# B&R Automation Studio project MotionTestBenchMaster (part 38)

#### Cyclic.sfc - Cyclic code
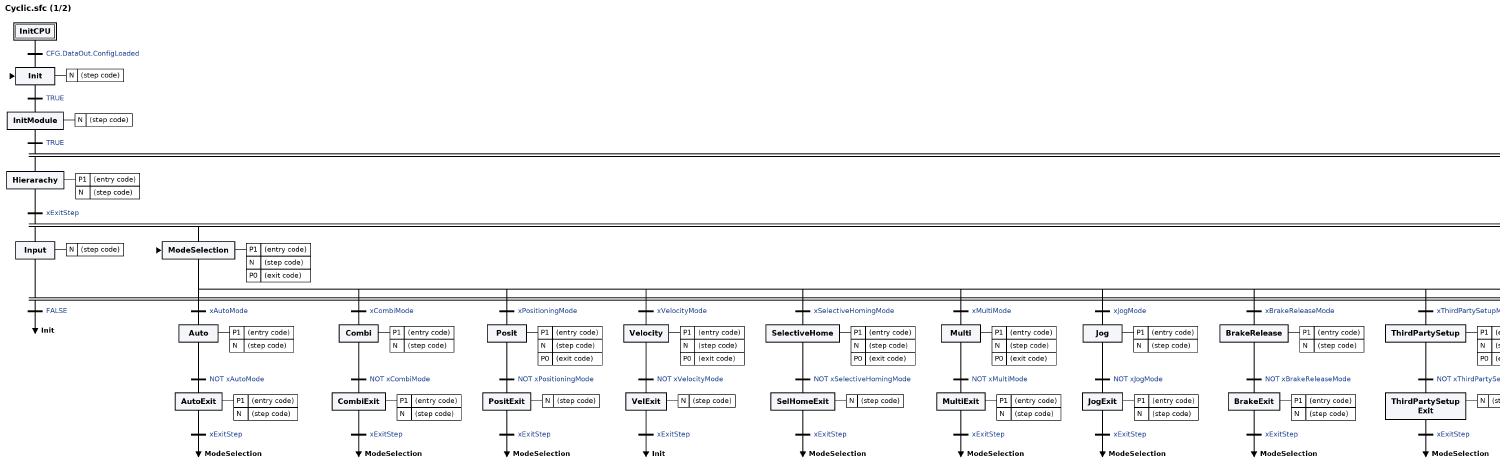
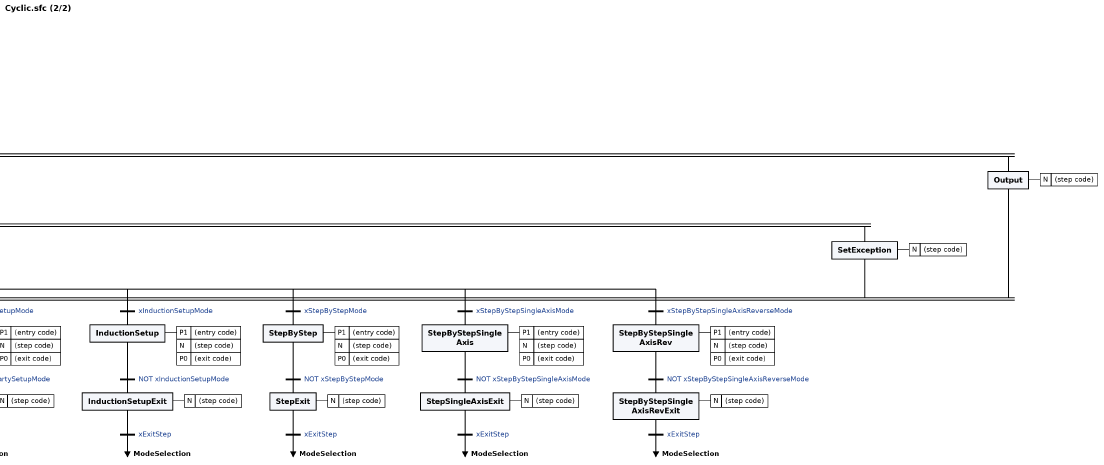
```iecst
PROGRAM _CYCLIC
INITIAL_STEP InitCPU:
END_STEP
TRANSITION FROM InitCPU TO Init:=
CFG.DataOut.ConfigLoaded
END_TRANSITION
STEP Init:
(* Pointer to master position *)
IF NOT CFG_MC.Generic.SyncroPar.ExternalEncoder THEN
	VAR_Machine.stMasterModule.iq_stParameters.i_pstMasterPositionStruct	:= ADR(ITC_Motion);	//VIRTUAL POSITION (SUPERCOMBI)
END_IF

// Init Encoder Emulation
fbEncoderEmulation.i_pstSrcAxis			:= ADR(VAR_AxFillerMain);
fbEncoderEmulation.i_pstEncEmulAxis		:= ADR(VAR_AxEncEmul);
IF CFG_MC.Generic.EmulationCardPulses > 0 THEN
	fbEncoderEmulation.i_uiNumberOfPulses	:= CFG_MC.Generic.EmulationCardPulses;
ELSE
	fbEncoderEmulation.i_uiNumberOfPulses	:= 1024;
END_IF
fbEncoderEmulation.i_xEnable			:= TRUE;
END_STEP
TRANSITION FROM Init TO InitModule:=
TRUE
END_TRANSITION
STEP InitModule:
MC_InputOutput;

(* Machine excpetion *)
fbQuickStopFromPlc.i_psAlarmName		:= ADR('PlcQuickStop');
fbQuickStopFromPlc.i_pstMpAlarmXLink	:= ADR(gMainAlarmXCoreLink);
fbQuickStopFromPlc.i_pxAcknowledge		:= ADR(VAR_Machine.iq_stCmd.i_xReset);
fbQuickStopFromPlc.i_pxInitCoreDone		:= ADR(VAR_Machine.stMasterModule.iq_stCmd.i_xAlarmInitOk);
fbQuickStopFromPlc.i_xAutoAck			:= TRUE;

fbKochModuleNotReady.i_psAlarmName		:= ADR('KochNotReady');
fbKochModuleNotReady.i_pstMpAlarmXLink	:= ADR(gMainAlarmXCoreLink);
fbKochModuleNotReady.i_pxAcknowledge	:= ADR(VAR_Machine.iq_stCmd.i_xReset);
fbKochModuleNotReady.i_pxInitCoreDone	:= ADR(VAR_Machine.stMasterModule.iq_stCmd.i_xAlarmInitOk);
fbKochModuleNotReady.i_xAutoAck			:= TRUE;

fbSeamerFanFault.i_psAlarmName			:= ADR('SeamerFanFault');
fbSeamerFanFault.i_pstMpAlarmXLink		:= ADR(gMainAlarmXCoreLink);
fbSeamerFanFault.i_pxAcknowledge		:= ADR(VAR_Machine.iq_stCmd.i_xReset);
fbSeamerFanFault.i_pxInitCoreDone		:= ADR(VAR_Machine.stMasterModule.iq_stCmd.i_xAlarmInitOk);
fbSeamerFanFault.i_xAutoAck				:= FALSE;
END_STEP
TRANSITION FROM InitModule TO (Hierarachy,Output):=
TRUE
END_TRANSITION
STEP Hierarachy:
IF 	VAR_Machine.stFillerModule.iq_stStatus.q_xInitDone	AND
	VAR_Machine.stInletModule.iq_stStatus.q_xInitDone 	AND
	VAR_Machine.stOutletModule.iq_stStatus.q_xInitDone	THEN

	xExitStep	:=	TRUE;

	// First and last real FILLER axis
	uiMinRealFillerIndex := CST_LastFillerModuleAxis;
	uiMaxRealFillerIndex := CST_FirstFillerModuleAxis;

	FOR uiAxisIndex := CST_FirstFillerModuleAxis TO CST_LastFillerModuleAxis DO
		IF VAR_Machine.stFillerModule.iq_astSubModuleAxis[uiAxisIndex].iq_stStatus.q_stMainAxisStatus.q_xAxisReal THEN
			uiMinRealFillerIndex := MIN(uiMinRealFillerIndex, uiAxisIndex);
			uiMaxRealFillerIndex := MAX(uiMaxRealFillerIndex, uiAxisIndex);
		END_IF
	END_FOR

	// Inlet module last axis homing position = filler module first axis act position
	uiMaxRealInletIndex := CST_FirstInletModuleAxis;
	IF VAR_Machine.stInletModule.iq_stStatus.q_xModuleReal	THEN
		FOR uiAxisIndex := CST_MainAxis TO CST_LastInletModuleAxis DO
			IF VAR_Machine.stInletModule.iq_astSubModuleAxis[uiAxisIndex].iq_stStatus.q_stMainAxisStatus.q_xAxisReal THEN
				uiMaxRealInletIndex := MAX(uiMaxRealInletIndex, uiAxisIndex);
			END_IF
		END_FOR
		IF uiMaxRealInletIndex <> CST_FirstInletModuleAxis THEN
			VAR_Machine.stInletModule.iq_astSubModuleAxis[uiMaxRealInletIndex].iq_stParam.i_udiHomingPosition	:=
				ADR(VAR_Machine.stFillerModule.iq_astSubModuleAxis[uiMinRealFillerIndex].iq_stStatus.q_stMainAxisStatus.q_lrPosition);
		END_IF
	END_IF

	// Outlet module first axis homing position = filler module last axis act position
	uiMinRealOutletIndex := CST_LastOutletModuleAxis;
	IF VAR_Machine.stOutletModule.iq_stStatus.q_xModuleReal	THEN
		FOR uiAxisIndex := CST_FirstOutletModuleAxis TO CST_MainAxis DO
			IF VAR_Machine.stOutletModule.iq_astSubModuleAxis[uiAxisIndex].iq_stStatus.q_stMainAxisStatus.q_xAxisReal THEN
				uiMinRealOutletIndex := MIN(uiMinRealOutletIndex, uiAxisIndex);
			END_IF
		END_FOR
		IF uiMinRealOutletIndex <> CST_LastOutletModuleAxis THEN
			VAR_Machine.stOutletModule.iq_astSubModuleAxis[uiMinRealOutletIndex].iq_stParam.i_udiHomingPosition	:=
				ADR(VAR_Machine.stFillerModule.iq_astSubModuleAxis[uiMaxRealFillerIndex].iq_stStatus.q_stMainAxisStatus.q_lrPosition);
		END_IF
	END_IF
END_IF

//NEW MANAGEMENT //FR
HMI_AxisIndex := 2;//0 is master
//HMI Crate array axis present and name
//INlet Module
IF VAR_Machine.stInletModule.iq_stStatus.q_xModuleReal THEN
	FOR uiAxisIndex := CST_FirstInletModuleAxis TO CST_LastInletModuleAxis DO
		IF VAR_Machine.stInletModule.iq_astSubModuleAxis[uiAxisIndex].iq_stStatus.q_stMainAxisStatus.q_xAxisReal THEN
			HMI_MC_GenericAxisDataNew[HMI_AxisIndex].xHmiPresent	:= TRUE;
			HMI_MC_GenericAxisDataNew[HMI_AxisIndex].uiAxisID		:= uiAxisIndex + CST_InletSubModuleHmiStart;
			HMI_AxisIndex := HMI_AxisIndex +1;
		END_IF
	END_FOR
END_IF
//HMI Crate array axis present and name
//Filler Module
IF VAR_Machine.stFillerModule.iq_stStatus.q_xModuleReal	THEN
	FOR uiAxisIndex := CST_FirstFillerModuleAxis TO CST_LastFillerModuleAxis DO
		IF VAR_Machine.stFillerModule.iq_astSubModuleAxis[uiAxisIndex].iq_stStatus.q_stMainAxisStatus.q_xAxisReal THEN
			HMI_MC_GenericAxisDataNew[HMI_AxisIndex].xHmiPresent	:= TRUE;
			HMI_MC_GenericAxisDataNew[HMI_AxisIndex].uiAxisID		:= uiAxisIndex + CST_FillerSubModuleHmiStart;
			HMI_AxisIndex := HMI_AxisIndex +1;
		END_IF
	END_FOR
END_IF
//HMI Crate array axis present and name
//Outlet Module
IF VAR_Machine.stOutletModule.iq_stStatus.q_xModuleReal	THEN
	FOR uiAxisIndex := CST_FirstOutletModuleAxis TO CST_LastOutletModuleAxis DO
		IF VAR_Machine.stOutletModule.iq_astSubModuleAxis[uiAxisIndex].iq_stStatus.q_stMainAxisStatus.q_xAxisReal THEN
			HMI_MC_GenericAxisDataNew[HMI_AxisIndex].xHmiPresent	:= TRUE;
			HMI_MC_GenericAxisDataNew[HMI_AxisIndex].uiAxisID		:= uiAxisIndex + CST_OutletSubModuleHmiStart;
			HMI_AxisIndex := HMI_AxisIndex +1;
		END_IF
	END_FOR
END_IF

FOR HMI_AxisIndex := 2 TO 14 DO //vrma

CASE HMI_MC_GenericAxisDataNew[HMI_AxisIndex].uiAxisID OF

	105:
		HMI_MC_GenericAxisDataNew[HMI_AxisIndex].usiHmiName	:= CFG_MC.Axes.Filler.In[10].HmiNameId;

	106:
		HMI_MC_GenericAxisDataNew[HMI_AxisIndex].usiHmiName	:= CFG_MC.Axes.Filler.In[9].HmiNameId;

	107:
		HMI_MC_GenericAxisDataNew[HMI_AxisIndex].usiHmiName	:= CFG_MC.Axes.Filler.In[8].HmiNameId;

	108:
		HMI_MC_GenericAxisDataNew[HMI_AxisIndex].usiHmiName	:= CFG_MC.Axes.Filler.In[7].HmiNameId;

	109:
		HMI_MC_GenericAxisDataNew[HMI_AxisIndex].usiHmiName	:= CFG_MC.Axes.Filler.In[6].HmiNameId;

	110:
		HMI_MC_GenericAxisDataNew[HMI_AxisIndex].usiHmiName	:= CFG_MC.Axes.Filler.In[5].HmiNameId;

	111:
		HMI_MC_GenericAxisDataNew[HMI_AxisIndex].usiHmiName	:= CFG_MC.Axes.Filler.In[4].HmiNameId;

	112:
		HMI_MC_GenericAxisDataNew[HMI_AxisIndex].usiHmiName	:= CFG_MC.Axes.Filler.In[3].HmiNameId;

	113:
		HMI_MC_GenericAxisDataNew[HMI_AxisIndex].usiHmiName	:= CFG_MC.Axes.Filler.In[2].HmiNameId;

	114:
		HMI_MC_GenericAxisDataNew[HMI_AxisIndex].usiHmiName	:= CFG_MC.Axes.Filler.In[1].HmiNameId;

	115:
		HMI_MC_GenericAxisDataNew[HMI_AxisIndex].usiHmiName	:= CFG_MC.Axes.Filler.Main.HmiNameId;

	116:
		HMI_MC_GenericAxisDataNew[HMI_AxisIndex].usiHmiName	:= CFG_MC.Axes.Filler.Out[1].HmiNameId;

	117:
		HMI_MC_GenericAxisDataNew[HMI_AxisIndex].usiHmiName	:= CFG_MC.Axes.Filler.Out[2].HmiNameId;

	118:
		HMI_MC_GenericAxisDataNew[HMI_AxisIndex].usiHmiName	:= CFG_MC.Axes.Filler.Out[3].HmiNameId;

	119:
		HMI_MC_GenericAxisDataNew[HMI_AxisIndex].usiHmiName	:= CFG_MC.Axes.Filler.Out[4].HmiNameId;

	120:
		HMI_MC_GenericAxisDataNew[HMI_AxisIndex].usiHmiName	:= CFG_MC.Axes.Filler.Out[5].HmiNameId;

	121:
		HMI_MC_GenericAxisDataNew[HMI_AxisIndex].usiHmiName	:= CFG_MC.Axes.Filler.Out[6].HmiNameId;

	211:
		HMI_MC_GenericAxisDataNew[HMI_AxisIndex].usiHmiName	:= CFG_MC.Axes.Inlet.In[4].HmiNameId;

	212:
		HMI_MC_GenericAxisDataNew[HMI_AxisIndex].usiHmiName	:= CFG_MC.Axes.Inlet.In[3].HmiNameId;

	213:
		HMI_MC_GenericAxisDataNew[HMI_AxisIndex].usiHmiName	:= CFG_MC.Axes.Inlet.In[2].HmiNameId;

	214:
		HMI_MC_GenericAxisDataNew[HMI_AxisIndex].usiHmiName	:= CFG_MC.Axes.Inlet.In[1].HmiNameId;

	215:
		HMI_MC_GenericAxisDataNew[HMI_AxisIndex].usiHmiName	:= CFG_MC.Axes.Inlet.Main.HmiNameId;

	216:
		HMI_MC_GenericAxisDataNew[HMI_AxisIndex].usiHmiName	:= CFG_MC.Axes.Inlet.Out[1].HmiNameId;

	217:
		HMI_MC_GenericAxisDataNew[HMI_AxisIndex].usiHmiName	:= CFG_MC.Axes.Inlet.Out[2].HmiNameId;

	218:
		HMI_MC_GenericAxisDataNew[HMI_AxisIndex].usiHmiName	:= CFG_MC.Axes.Inlet.Out[3].HmiNameId;

	219:
		HMI_MC_GenericAxisDataNew[HMI_AxisIndex].usiHmiName	:= CFG_MC.Axes.Inlet.Out[4].HmiNameId;

	311:
		HMI_MC_GenericAxisDataNew[HMI_AxisIndex].usiHmiName	:= CFG_MC.Axes.Outlet.In[4].HmiNameId;

	312:
		HMI_MC_GenericAxisDataNew[HMI_AxisIndex].usiHmiName	:= CFG_MC.Axes.Outlet.In[3].HmiNameId;

	313:
		HMI_MC_GenericAxisDataNew[HMI_AxisIndex].usiHmiName	:= CFG_MC.Axes.Outlet.In[2].HmiNameId;

	314:
		HMI_MC_GenericAxisDataNew[HMI_AxisIndex].usiHmiName	:= CFG_MC.Axes.Outlet.In[1].HmiNameId;

	315:
		HMI_MC_GenericAxisDataNew[HMI_AxisIndex].usiHmiName	:= CFG_MC.Axes.Outlet.Main.HmiNameId;

	316:
		HMI_MC_GenericAxisDataNew[HMI_AxisIndex].usiHmiName	:= CFG_MC.Axes.Outlet.Out[1].HmiNameId;

	317:
		HMI_MC_GenericAxisDataNew[HMI_AxisIndex].usiHmiName	:= CFG_MC.Axes.Outlet.Out[2].HmiNameId;

	318:
		HMI_MC_GenericAxisDataNew[HMI_AxisIndex].usiHmiName	:= CFG_MC.Axes.Outlet.Out[3].HmiNameId;

	319:
		HMI_MC_GenericAxisDataNew[HMI_AxisIndex].usiHmiName	:= CFG_MC.Axes.Outlet.Out[4].HmiNameId;
	ELSE
		HMI_MC_GenericAxisDataNew[HMI_AxisIndex].usiHmiName		:= 0;
END_CASE

END_FOR
END_STEP
ENTRY_ACTION
xExitStep	:=	FALSE;

VAR_Machine.stMasterModule.iq_stCmd.i_xMachineInitDone	:=	TRUE;
VAR_Machine.stFillerModule.iq_stCmd.i_xMachineInitDone	:=	TRUE;
VAR_Machine.stInletModule.iq_stCmd.i_xMachineInitDone	:=	TRUE;
VAR_Machine.stOutletModule.iq_stCmd.i_xMachineInitDone	:=	TRUE;
END_ACTION
TRANSITION FROM Hierarachy TO (Input,ModeSelection,SetException):=
xExitStep
END_TRANSITION
STEP Input:
(* Input Signals *)
xInputJog							:= VAR_Machine.iq_stCmd.i_xJogMode;
xInputAuto							:= VAR_Machine.iq_stCmd.i_xAuto	AND NOT VAR_Machine.iq_stCmd.i_xStepByStep AND NOT VAR_Machine.iq_stCmd.i_xStepByStepSingleAxis AND NOT VAR_Machine.iq_stCmd.i_xStepByStepSingleAxisReverse;//v999
xInputCombi							:= VAR_Machine.iq_stCmd.i_xCombi;
xInputMulti							:= VAR_Machine.iq_stCmd.i_xMulti;
xInputSelHoming						:= VAR_Machine.iq_stCmd.i_xSelectiveHoming;
xInputPositioning					:= VAR_Machine.iq_stCmd.i_xPositioning;
xInputBrakeRelease					:= VAR_Machine.iq_stCmd.i_xBrakeRelease;
xInputVelocity						:= VAR_Machine.iq_stCmd.i_xVelocity;
xInputStepByStep					:= VAR_Machine.iq_stCmd.i_xAuto AND VAR_Machine.iq_stCmd.i_xStepByStep;
xInputStepByStepSingleAxis			:= (VAR_Machine.iq_stCmd.i_xAuto AND VAR_Machine.iq_stCmd.i_xStepByStepSingleAxis) OR (NOT VAR_Machine.iq_stCmd.i_xAuto AND VAR_Machine.iq_stCmd.i_xStepByStepSingleAxis);//V4.A.A.1.7.0 FootBar
xInputStepByStepSingleAxisRev		:= (VAR_Machine.iq_stCmd.i_xAuto AND VAR_Machine.iq_stCmd.i_xStepByStepSingleAxisReverse) OR (NOT VAR_Machine.iq_stCmd.i_xAuto AND VAR_Machine.iq_stCmd.i_xStepByStepSingleAxisReverse);//v999
xInputThirdPartySetup				:= VAR_Machine.iq_stCmd.i_xThirdPartySetup;
xInputInductionSetup				:= VAR_Machine.iq_stCmd.i_xInductionSetup;

(* Acceleration and deceleration calculation *)
IF 	rOldAccelerationValue <> MC_InputOutput.Network.Machine.Parameters.AutoAccelerationTime 	AND
	MC_InputOutput.Network.Machine.Parameters.AutoAccelerationTime > 0						  	AND
	MC_InputOutput.Network.Machine.Status.MachineMaxSpeed	> 0									THEN

	VAR_Machine.stMasterModule.iq_stParameters.i_rEndlessAcceleration
		:= FC_GetAccFromTimeAndJerk(	MC_InputOutput.Network.Machine.Parameters.AutoAccelerationTime,
								 		CFG_MC.Movements.Jerk,
										MC_InputOutput.Network.Machine.Status.MachineMaxSpeed / 10.0);

	VAR_Machine.stMasterModule.iq_stParameters.i_rEndlessAcceleration
		:= MIN(VAR_Machine.stMasterModule.iq_stParameters.i_rEndlessAcceleration, VAR_EmergencyDec);

	VAR_Machine.stFillerModule.iq_stParameters.i_rEndlessAcceleration
		:= VAR_Machine.stMasterModule.iq_stParameters.i_rEndlessAcceleration;

	VAR_Machine.stInletModule.iq_stParameters.i_rEndlessAcceleration
		:= VAR_Machine.stMasterModule.iq_stParameters.i_rEndlessAcceleration;

	VAR_Machine.stOutletModule.iq_stParameters.i_rEndlessAcceleration
		:= VAR_Machine.stMasterModule.iq_stParameters.i_rEndlessAcceleration;

	rOldAccelerationValue := MC_InputOutput.Network.Machine.Parameters.AutoAccelerationTime;
END_IF

IF 	rOldDecelerationValue <> MC_InputOutput.Network.Machine.Parameters.AutoDecelerationTime 	AND
	MC_InputOutput.Network.Machine.Parameters.AutoDecelerationTime 	> 0					  		AND
	MC_InputOutput.Network.Machine.Status.MachineMaxSpeed			> 0							THEN

	VAR_Machine.stMasterModule.iq_stParameters.i_rEndlessDeceleration
		:= FC_GetAccFromTimeAndJerk(	MC_InputOutput.Network.Machine.Parameters.AutoDecelerationTime,
										CFG_MC.Movements.Jerk,
										MC_InputOutput.Network.Machine.Status.MachineMaxSpeed / 10.0);

	VAR_Machine.stMasterModule.iq_stParameters.i_rEndlessDeceleration
		:= MIN(VAR_Machine.stMasterModule.iq_stParameters.i_rEndlessDeceleration, VAR_EmergencyDec);

	VAR_Machine.stFillerModule.iq_stParameters.i_rEndlessDeceleration
		:= VAR_Machine.stMasterModule.iq_stParameters.i_rEndlessDeceleration;

	VAR_Machine.stInletModule.iq_stParameters.i_rEndlessDeceleration
		:= VAR_Machine.stMasterModule.iq_stParameters.i_rEndlessDeceleration;

	VAR_Machine.stOutletModule.iq_stParameters.i_rEndlessDeceleration
		:= VAR_Machine.stMasterModule.iq_stParameters.i_rEndlessDeceleration;

	rOldDecelerationValue := MC_InputOutput.Network.Machine.Parameters.AutoDecelerationTime;
END_IF

(* Enable curves *)
VAR_Machine.stMasterModule.iq_stCmd.i_xEnableCurves	:=	MC_InputOutput.Network.Machine.Commands.MasterEncoderPositionValid; //COMBI

(* Input from safety system *)
VAR_Machine.stFillerModule.iq_stCmd.i_xEnable	:= MC_InputOutput.Safety.Filler.Commands.EnableModule;
VAR_Machine.stInletModule.iq_stCmd.i_xEnable	:= MC_InputOutput.Safety.Inlet.Commands.EnableModule;
VAR_Machine.stOutletModule.iq_stCmd.i_xEnable	:= MC_InputOutput.Safety.Outlet.Commands.EnableModule;

xSlowMotionCommandOutletForward		:= MC_InputOutput.Network.Outlet.Commands.SlowMotionForward;
xSlowMotionCommandOutletBackward	:= MC_InputOutput.Network.Outlet.Commands.SlowMotionBackward;
xSlowMotionCommandOutlet			:= xSlowMotionCommandOutletForward OR xSlowMotionCommandOutletBackward;

xSlowMotionCommandInletForward		:= MC_InputOutput.Network.Inlet.Commands.SlowMotionForward;
xSlowMotionCommandInletBackward		:= MC_InputOutput.Network.Inlet.Commands.SlowMotionBackward;
xSlowMotionCommandInlet				:= xSlowMotionCommandInletForward OR xSlowMotionCommandInletBackward;
END_STEP
STEP ModeSelection:
xModeReady	:= NOT xAutoMode AND NOT xPositioningMode AND NOT xSelectiveHomingMode	AND NOT xJogMode AND NOT xPositioningMode AND NOT xThirdPartySetupMode AND NOT xInductionSetupMode AND
				(NOT tofReactionActive.Q OR	xInputMulti OR xInputStepByStepSingleAxis);//V1.7.2

xNoOpActive				:= TRUE;
xAutoActive				:= FALSE;
xBrakeReleaseActive		:= FALSE;
xPositioningActive		:= FALSE;
xSelHomingActive		:= FALSE;
xJogActive				:= FALSE;
xMultiActive			:= FALSE;
xVelocityActive			:= FALSE;
xStepByStepActive		:= FALSE;
xStepByStepSingleAxisActive	:= FALSE;//V4.A.A.1.7.0
xStepByStepSingleAxisRevActive	:= FALSE; //v999
xCombiActive			:= FALSE;
xThirdPartySetupActive	:= FALSE;
xInductionSetupActive	:= FALSE;

IF xModeReady THEN
	IF xInputAuto THEN
		xAutoMode					:= TRUE;
	ELSIF xInputCombi THEN
		xCombiMode					:= TRUE;
	ELSIF xInputPositioning THEN
		xPositioningMode			:= TRUE;
	ELSIF xInputSelHoming THEN
		xSelectiveHomingMode		:= TRUE;
	ELSIF xInputJog THEN
		xJogMode					:= TRUE;
	ELSIF xInputMulti THEN
		xMultiMode					:= TRUE;
	ELSIF xInputVelocity THEN
		xVelocityMode				:= TRUE;
	ELSIF xInputStepByStep THEN
		xStepByStepMode				:= TRUE;
	ELSIF xInputStepByStepSingleAxis THEN//V4.A.A.1.7.0
		xStepByStepSingleAxisMode	:= TRUE;//V4.A.A.1.7.0
	ELSIF xInputStepByStepSingleAxisRev THEN//v999
		xStepByStepSingleAxisReverseMode := TRUE;//v999
	ELSIF xInputThirdPartySetup THEN
		xThirdPartySetupMode		:= TRUE;
	ELSIF xInputInductionSetup THEN
		xInductionSetupMode			:= TRUE;
	END_IF
ELSIF tofReactionActive.Q AND xInputBrakeRelease THEN
	xBrakeReleaseMode			:= TRUE;
END_IF
END_STEP
ENTRY_ACTION
xExitStep	:= FALSE;

VAR_Machine.stMasterModule.iq_stCmd.i_xStart	:= FALSE;
VAR_Machine.stFillerModule.iq_stCmd.i_xStart	:= FALSE;
VAR_Machine.stInletModule.iq_stCmd.i_xStart		:= FALSE;
VAR_Machine.stOutletModule.iq_stCmd.i_xStart	:= FALSE;

// For safety reason all bits are set to FALSE
xJogMode 							:= FALSE;
xAutoMode 							:= FALSE;
xMultiMode 							:= FALSE;
xPositioningMode 					:= FALSE;
xSelectiveHomingMode				:= FALSE;
xVelocityMode						:= FALSE;
xCombiMode							:= FALSE;
xBrakeReleaseMode					:= FALSE;
xStepByStepMode						:= FALSE;
xStepByStepSingleAxisMode			:= FALSE;//V4.A.A.1.7.0 Footbar
xStepByStepSingleAxisReverseMode	:= FALSE;//V999
xThirdPartySetupMode				:= FALSE;
xInductionSetupMode					:= FALSE;
END_ACTION
EXIT_ACTION
xNoOpActive	:= FALSE;
END_ACTION
TRANSITION FROM ModeSelection TO Auto:=
xAutoMode
END_TRANSITION
TRANSITION FROM ModeSelection TO Combi:=
xCombiMode
END_TRANSITION
STEP Combi:
IF xReactionActive	OR NOT xInputCombi	THEN
	xCombiMode	:=	FALSE;
END_IF

xCombiActive	:= TRUE;

CASE uiCombiStep OF
	0:
		xCombiSynchronized		:=	FALSE;
		xCombiSynchroStopDone	:=	FALSE;
		xCombiFixedSpeed		:=	FALSE;
		xCombiSynchroInProgress	:=	FALSE;

		VAR_Machine.stFillerModule.iq_stCmd.i_xAutoMode	:=	TRUE;
		VAR_Machine.stOutletModule.iq_stCmd.i_xAutoMode	:=	VAR_Machine.stOutletModule.iq_stStatus.q_xModuleReal;
		VAR_Machine.stInletModule.iq_stCmd.i_xAutoMode	:=	VAR_Machine.stInletModule.iq_stStatus.q_xModuleReal;

		uiCombiStep	:=	40;

	40:
		IF 	VAR_Machine.stFillerModule.iq_stStatus.q_xAutoActive	AND
			(VAR_Machine.stOutletModule.iq_stStatus.q_xAutoActive	OR NOT
			VAR_Machine.stOutletModule.iq_stStatus.q_xModuleReal)	AND
			(VAR_Machine.stInletModule.iq_stStatus.q_xAutoActive	OR NOT
			VAR_Machine.stInletModule.iq_stStatus.q_xModuleReal)	THEN

			IF 	NOT VAR_Machine.stFillerModule.iq_stStatus.q_xSynchroWithOffset		AND
				NOT VAR_Machine.stOutletModule.iq_stStatus.q_xSynchroWithOffset		AND
				NOT VAR_Machine.stInletModule.iq_stStatus.q_xSynchroWithOffset		THEN

				VAR_Machine.stMasterModule.iq_stParameters.i_lrRephasingPosition	:=
					FC_RephasingMachine(iq_astInletSubModuleAxis	:=	VAR_Machine.stInletModule.iq_astSubModuleAxis,
										iq_astFillerSubModuleAxis	:=	VAR_Machine.stFillerModule.iq_astSubModuleAxis,
										iq_astOutletSubModuleAxis	:=	VAR_Machine.stOutletModule.iq_astSubModuleAxis);

				VAR_Machine.stFillerModule.iq_stParameters.i_lrRephasingPosition
					:=	VAR_Machine.stMasterModule.iq_stParameters.i_lrRephasingPosition;

				VAR_Machine.stOutletModule.iq_stParameters.i_lrRephasingPosition
					:=	VAR_Machine.stMasterModule.iq_stParameters.i_lrRephasingPosition;

				VAR_Machine.stInletModule.iq_stParameters.i_lrRephasingPosition
					:=	VAR_Machine.stMasterModule.iq_stParameters.i_lrRephasingPosition;

				uiCombiStep	:=	100;
			END_IF
		END_IF

	100:(* Wait Master Rephased *)
		VAR_Machine.stMasterModule.iq_stCmd.i_xCombi					:=	TRUE;
		VAR_Machine.stMasterModule.iq_stCmd.i_xMasterRephasingRequest	:= 	TRUE;

		IF VAR_Machine.stMasterModule.iq_stStatus.q_xCombiActive AND VAR_Machine.stMasterModule.iq_stStatus.q_xMasterRephased THEN
			VAR_Machine.stMasterModule.iq_stCmd.i_xMasterRephasingRequest	:= 	FALSE;
			uiCombiStep	:=	110;
		END_IF

	110:(* Wait for start Signal *)
		IF VAR_Machine.iq_stCmd.i_xStart THEN
			VAR_Machine.stFillerModule.iq_stCmd.i_xStart	:=	TRUE;
			VAR_Machine.stOutletModule.iq_stCmd.i_xStart	:=	VAR_Machine.stOutletModule.iq_stStatus.q_xModuleReal;
			VAR_Machine.stInletModule.iq_stCmd.i_xStart		:=	VAR_Machine.stInletModule.iq_stStatus.q_xModuleReal;
			uiCombiStep	:=	120;
		END_IF

	120:(* Wait for submodules synchronized *)
		IF VAR_Machine.stFillerModule.iq_stStatus.q_xRealAxesSynchronized		AND
			VAR_Machine.stFillerModule.iq_stStatus.q_xAutoActive				AND
			VAR_Machine.stFillerModule.iq_stStatus.q_xMasterRephased			AND

			((VAR_Machine.stOutletModule.iq_stStatus.q_xRealAxesSynchronized	AND
			VAR_Machine.stOutletModule.iq_stStatus.q_xMasterRephased			AND
			VAR_Machine.stOutletModule.iq_stStatus.q_xAutoActive)				OR NOT
			VAR_Machine.stOutletModule.iq_stStatus.q_xModuleReal)				AND

			((VAR_Machine.stInletModule.iq_stStatus.q_xRealAxesSynchronized		AND
			VAR_Machine.stInletModule.iq_stStatus.q_xMasterRephased				AND
			VAR_Machine.stInletModule.iq_stStatus.q_xAutoActive)				OR NOT
			VAR_Machine.stInletModule.iq_stStatus.q_xModuleReal)				THEN

			VAR_Machine.stMasterModule.iq_stCmd.i_xStart	:=	TRUE;
			xEncEmulationEnable	:= TRUE;
			uiCombiStep	:=	130;
		END_IF

	130:(* Wait for master synchronized with the external reference *)
		xCombiSynchroInProgress	:=	TRUE;

		IF NOT VAR_Machine.iq_stCmd.i_xStart THEN
			VAR_Machine.stMasterModule.iq_stCmd.i_xCombiSynchroStop	:=	TRUE;
			uiCombiStep	:=	150;
		ELSIF VAR_Machine.stMasterModule.iq_stStatus.q_xModuleSynchronized THEN
			uiCombiStep	:=	140;
		END_IF

	140:(* Module synchronized with the master *)
		xCombiSynchroInProgress	:=	FALSE;
		xCombiSynchronized		:=	TRUE;
		xCombiSynchroStopDone	:=	FALSE;
		xCombiFixedSpeed		:=	FALSE;

		IF NOT VAR_Machine.iq_stCmd.i_xStart OR VAR_Machine.iq_stCmd.i_xCombiSynchroStop THEN
			xCombiSynchroInProgress	:=	FALSE;
			xCombiSynchronized		:=	FALSE;
			xCombiSynchroStopDone	:=	TRUE;
			xCombiFixedSpeed		:=	FALSE;

			VAR_Machine.stMasterModule.iq_stCmd.i_xCombiSynchroStop	:=	TRUE;
			uiCombiStep		:=	150;
		ELSIF VAR_Machine.iq_stCmd.i_xOnePitchShift	THEN
			uiCombiStep		:=	600;
		ELSIF VAR_Machine.iq_stCmd.i_xAxisPhaseShift THEN
			IF VAR_Machine.iq_stParameter.i_uiAxisSelected >= CST_FillerSubModuleHmiStart AND
				VAR_Machine.iq_stParameter.i_uiAxisSelected <= CST_FillerSubModuleHmiStart + CST_LastFillerModuleAxis	THEN

				VAR_Machine.stFillerModule.iq_stParameters.i_uiAxisSelected
					:=	VAR_Machine.iq_stParameter.i_uiAxisSelected - CST_FillerSubModuleHmiStart;

				VAR_Machine.stFillerModule.iq_stParameters.i_rPhaseShiftDistance
					:=	LREAL_TO_REAL(FC_TeensOfmmToDegrees(VAR_Machine.iq_stParameter.i_iAxisPhaseShiftDistance, CFG_MC.Mechanical.MachineStep, TRUE, FALSE));

				uiCombiStep	:=	200;
			ELSIF VAR_Machine.iq_stParameter.i_uiAxisSelected >= CST_OutletSubModuleHmiStart AND
				VAR_Machine.iq_stParameter.i_uiAxisSelected <= CST_OutletSubModuleHmiStart + CST_LastOutletModuleAxis THEN

				VAR_Machine.stOutletModule.iq_stParameters.i_uiAxisSelected
					:=	VAR_Machine.iq_stParameter.i_uiAxisSelected - CST_OutletSubModuleHmiStart;

				VAR_Machine.stOutletModule.iq_stParameters.i_rPhaseShiftDistance
					:=	LREAL_TO_REAL(FC_TeensOfmmToDegrees(VAR_Machine.iq_stParameter.i_iAxisPhaseShiftDistance, CFG_MC.Mechanical.MachineStep, TRUE, FALSE));

				uiCombiStep	:=	300;
			ELSIF VAR_Machine.iq_stParameter.i_uiAxisSelected >= CST_InletSubModuleHmiStart AND
				VAR_Machine.iq_stParameter.i_uiAxisSelected <= CST_InletSubModuleHmiStart + CST_LastInletModuleAxis THEN

				VAR_Machine.stInletModule.iq_stParameters.i_uiAxisSelected
					:=	VAR_Machine.iq_stParameter.i_uiAxisSelected - CST_InletSubModuleHmiStart;

				VAR_Machine.stInletModule.iq_stParameters.i_rPhaseShiftDistance
					:=	LREAL_TO_REAL(FC_TeensOfmmToDegrees(VAR_Machine.iq_stParameter.i_iAxisPhaseShiftDistance, CFG_MC.Mechanical.MachineStep, TRUE, FALSE));

				uiCombiStep	:=	400;
			ELSIF VAR_Machine.iq_stParameter.i_uiAxisSelected = CST_MachinePhasingOffset THEN

				VAR_Machine.stMasterModule.iq_stParameters.i_uiAxisSelected
					:=	VAR_Machine.iq_stParameter.i_uiAxisSelected;

				VAR_Machine.stMasterModule.iq_stParameters.i_rPhaseShiftDistance
					:=	LREAL_TO_REAL(FC_TeensOfmmToDegrees(VAR_Machine.iq_stParameter.i_iAxisPhaseShiftDistance, CFG_MC.Mechanical.MachineStep, TRUE, FALSE));

				uiCombiStep	:=	700;
			END_IF
		END_IF

	150:(* Check Start Signal *)
		xCombiSynchroInProgress	:=	FALSE;
		xCombiSynchronized		:=	FALSE;
		xCombiSynchroStopDone	:=	TRUE;
		xCombiFixedSpeed		:=	TRUE;

		IF NOT VAR_Machine.iq_stCmd.i_xStart AND
			(VAR_Machine.stMasterModule.iq_stStatus.q_xCombiSynchroStopDone OR
			(VAR_Machine.stMasterModule.iq_stStatus.q_xModuleStopped 		AND NOT VAR_Machine.stMasterModule.iq_stStatus.q_xModuleSynchronized))	THEN

			VAR_Machine.stMasterModule.iq_stCmd.i_xCombiSynchroStop	:=	FALSE;
			VAR_Machine.stMasterModule.iq_stCmd.i_xStart			:=	FALSE;
			uiCombiStep	:=	160;
		END_IF

	160:(* Check Machine Stopped *)
		IF VAR_Machine.iq_stStatus.q_xMachineStopped THEN
			xCombiSynchroInProgress	:=	FALSE;
			xCombiSynchronized		:=	FALSE;
			xCombiSynchroStopDone	:=	FALSE;
			xCombiFixedSpeed		:=	FALSE;
			xEncEmulationEnable		:= FALSE;

			IF VAR_Machine.iq_stCmd.i_xStart AND NOT VAR_Machine.stMasterModule.iq_stStatus.q_xCombiSynchroStopDone THEN
				uiCombiStep	:=	120;
			ELSIF VAR_Machine.stMasterModule.iq_stStatus.q_xSynchroWithOffset		OR
					VAR_Machine.stFillerModule.iq_stStatus.q_xSynchroWithOffset		OR
					(VAR_Machine.stOutletModule.iq_stStatus.q_xSynchroWithOffset	AND
					VAR_Machine.stOutletModule.iq_stStatus.q_xModuleReal)			OR
					(VAR_Machine.stInletModule.iq_stStatus.q_xSynchroWithOffset		AND
					VAR_Machine.stInletModule.iq_stStatus.q_xModuleReal)			THEN

					uiCombiStep	:= 800;
			END_IF
		END_IF

	200:
		VAR_Machine.stFillerModule.iq_stCmd.i_xPhaseShift	:= TRUE;
		uiCombiStep	:= 210;

	210:
		IF NOT VAR_Machine.iq_stCmd.i_xStart OR VAR_Machine.iq_stCmd.i_xCombiSynchroStop THEN
			VAR_Machine.stMasterModule.iq_stCmd.i_xCombiSynchroStop	:=	TRUE;
		END_IF

		IF VAR_Machine.stFillerModule.iq_stStatus.q_xPhaseShiftDone AND NOT VAR_Machine.iq_stCmd.i_xAxisPhaseShift THEN
			VAR_Machine.stFillerModule.iq_stCmd.i_xPhaseShift	:= FALSE;

			IF VAR_Machine.stMasterModule.iq_stCmd.i_xCombiSynchroStop THEN
				uiCombiStep	:= 150;
			ELSE
				uiCombiStep	:= 140;
			END_IF
		END_IF

	300:
		VAR_Machine.stOutletModule.iq_stCmd.i_xPhaseShift	:= TRUE;
		uiCombiStep	:= 310;

	310:
		IF NOT VAR_Machine.iq_stCmd.i_xStart OR VAR_Machine.iq_stCmd.i_xCombiSynchroStop THEN
			VAR_Machine.stMasterModule.iq_stCmd.i_xCombiSynchroStop	:=	TRUE;
		END_IF;

		IF VAR_Machine.stOutletModule.iq_stStatus.q_xPhaseShiftDone AND NOT VAR_Machine.iq_stCmd.i_xAxisPhaseShift THEN
			VAR_Machine.stOutletModule.iq_stCmd.i_xPhaseShift	:= FALSE;

			IF VAR_Machine.stMasterModule.iq_stCmd.i_xCombiSynchroStop THEN
				uiCombiStep	:= 150;
			ELSE
				uiCombiStep	:= 140;
			END_IF
		END_IF

	400:
		VAR_Machine.stInletModule.iq_stCmd.i_xPhaseShift	:= TRUE;
		uiCombiStep	:= 410;

	410:
		IF NOT VAR_Machine.iq_stCmd.i_xStart OR VAR_Machine.iq_stCmd.i_xCombiSynchroStop THEN
			VAR_Machine.stMasterModule.iq_stCmd.i_xCombiSynchroStop	:=	TRUE;
		END_IF

		IF VAR_Machine.stInletModule.iq_stStatus.q_xPhaseShiftDone AND NOT VAR_Machine.iq_stCmd.i_xAxisPhaseShift THEN
			VAR_Machine.stInletModule.iq_stCmd.i_xPhaseShift	:= FALSE;

			IF VAR_Machine.stMasterModule.iq_stCmd.i_xCombiSynchroStop THEN
				uiCombiStep	:= 150;
			ELSE
				uiCombiStep	:= 140;
			END_IF
		END_IF

	600:(* One pitch shift *)
		VAR_Machine.stMasterModule.iq_stCmd.i_xOnePitchShift 	:=	TRUE;
		uiCombiStep	:= 610;

	610:
		VAR_Machine.iq_stStatus.q_xOnePitchShiftDone	:= VAR_Machine.stMasterModule.iq_stStatus.q_xOnePitchShifDone;

		IF NOT VAR_Machine.iq_stCmd.i_xStart OR VAR_Machine.iq_stCmd.i_xCombiSynchroStop THEN
			VAR_Machine.stMasterModule.iq_stCmd.i_xCombiSynchroStop	:=	TRUE;
			VAR_Machine.stMasterModule.iq_stCmd.i_xOnePitchShift 	:=	FALSE;
			VAR_Machine.iq_stStatus.q_xOnePitchShiftDone			:=	FALSE;
			uiCombiStep	:= 150;
		ELSIF (VAR_Machine.stMasterModule.iq_stStatus.q_xOnePitchShifDone AND NOT VAR_Machine.iq_stCmd.i_xOnePitchShift) THEN
			VAR_Machine.stMasterModule.iq_stCmd.i_xOnePitchShift	:= FALSE;
			uiCombiStep	:= 140;
		END_IF

	700:
		VAR_Machine.stMasterModule.iq_stCmd.i_xPhaseShift	:= TRUE;
		uiCombiStep	:= 710;

	710:
		IF NOT VAR_Machine.iq_stCmd.i_xStart OR VAR_Machine.iq_stCmd.i_xCombiSynchroStop THEN
			VAR_Machine.stMasterModule.iq_stCmd.i_xCombiSynchroStop	:=	TRUE;
		END_IF

		IF VAR_Machine.stMasterModule.iq_stStatus.q_xPhaseShiftDone AND NOT VAR_Machine.iq_stCmd.i_xAxisPhaseShift THEN
			VAR_Machine.stMasterModule.iq_stCmd.i_xPhaseShift	:= FALSE;
			IF VAR_Machine.stMasterModule.iq_stCmd.i_xCombiSynchroStop THEN
				uiCombiStep	:= 150;
			ELSE
				uiCombiStep	:= 140;
			END_IF
		END_IF

	800:
		VAR_Machine.stMasterModule.iq_stCmd.i_xPhaseCompensation	:= VAR_Machine.stMasterModule.iq_stStatus.q_xSynchroWithOffset;
		VAR_Machine.stFillerModule.iq_stCmd.i_xPhaseCompensation	:= VAR_Machine.stFillerModule.iq_stStatus.q_xSynchroWithOffset;
		VAR_Machine.stInletModule.iq_stCmd.i_xPhaseCompensation		:= VAR_Machine.stInletModule.iq_stStatus.q_xSynchroWithOffset;
		VAR_Machine.stOutletModule.iq_stCmd.i_xPhaseCompensation	:= VAR_Machine.stOutletModule.iq_stStatus.q_xSynchroWithOffset;

		uiCombiStep	:= 810;

	810:
		IF NOT VAR_Machine.stMasterModule.iq_stStatus.q_xSynchroWithOffset	AND
			NOT VAR_Machine.stFillerModule.iq_stStatus.q_xSynchroWithOffset	AND
			(NOT VAR_Machine.stOutletModule.iq_stStatus.q_xSynchroWithOffset OR
			NOT VAR_Machine.stOutletModule.iq_stStatus.q_xModuleReal)		AND
			(NOT VAR_Machine.stOutletModule.iq_stStatus.q_xSynchroWithOffset OR
			NOT VAR_Machine.stOutletModule.iq_stStatus.q_xModuleReal)		THEN

			VAR_Machine.stMasterModule.iq_stCmd.i_xPhaseCompensation	:= FALSE;
			VAR_Machine.stFillerModule.iq_stCmd.i_xPhaseCompensation	:= FALSE;
			VAR_Machine.stInletModule.iq_stCmd.i_xPhaseCompensation		:= FALSE;
			VAR_Machine.stOutletModule.iq_stCmd.i_xPhaseCompensation	:= FALSE;

			uiCombiStep	:= 160;
		END_IF
END_CASE
END_STEP
ENTRY_ACTION
uiCombiStep	:=	0;

xCombiSynchronized		:=	FALSE;
xCombiSynchroStopDone	:=	FALSE;
xCombiFixedSpeed		:=	FALSE;
xCombiSynchroInProgress	:=	FALSE;

VAR_Machine.stMasterModule.iq_stCmd.i_xCombiSynchroStop	:=	FALSE;
END_ACTION
TRANSITION FROM Combi TO CombiExit:=
NOT xCombiMode
END_TRANSITION
STEP CombiExit:
IF	NOT VAR_Machine.stMasterModule.iq_stStatus.q_xCombiActive	AND
	NOT VAR_Machine.stFillerModule.iq_stStatus.q_xAutoActive	AND
	(NOT VAR_Machine.stInletModule.iq_stStatus.q_xAutoActive	OR NOT
	VAR_Machine.stInletModule.iq_stStatus.q_xModuleReal)		AND
	(NOT VAR_Machine.stOutletModule.iq_stStatus.q_xAutoActive	OR NOT
	VAR_Machine.stOutletModule.iq_stStatus.q_xModuleReal)	THEN

	xExitStep	:= TRUE;
END_IF
END_STEP
ENTRY_ACTION
VAR_Machine.stFillerModule.iq_stCmd.i_xPhaseShift	:= FALSE;
VAR_Machine.stOutletModule.iq_stCmd.i_xPhaseShift	:= FALSE;
VAR_Machine.stInletModule.iq_stCmd.i_xPhaseShift	:= FALSE;

VAR_Machine.stMasterModule.iq_stCmd.i_xStart	:= FALSE;
VAR_Machine.stFillerModule.iq_stCmd.i_xStart	:= FALSE;
VAR_Machine.stOutletModule.iq_stCmd.i_xStart	:= FALSE;
VAR_Machine.stInletModule.iq_stCmd.i_xStart		:= FALSE;

VAR_Machine.stMasterModule.iq_stCmd.i_xCombi	:= FALSE;
VAR_Machine.stFillerModule.iq_stCmd.i_xAutoMode	:= FALSE;
VAR_Machine.stOutletModule.iq_stCmd.i_xAutoMode	:= FALSE;
VAR_Machine.stInletModule.iq_stCmd.i_xAutoMode	:= FALSE;

VAR_Machine.stMasterModule.iq_stCmd.i_xMasterRephasingRequest	:= FALSE;

VAR_Machine.stMasterModule.iq_stCmd.i_xPhaseCompensation	:= FALSE;
VAR_Machine.stFillerModule.iq_stCmd.i_xPhaseCompensation	:= FALSE;
VAR_Machine.stOutletModule.iq_stCmd.i_xPhaseCompensation	:= FALSE;
VAR_Machine.stInletModule.iq_stCmd.i_xPhaseCompensation		:= FALSE;

VAR_Machine.stMasterModule.iq_stCmd.i_xOnePitchShift 	:= FALSE;
VAR_Machine.iq_stStatus.q_xOnePitchShiftDone			:= FALSE;

xCombiSynchronized		:= FALSE;
xCombiSynchroStopDone	:= FALSE;
xCombiFixedSpeed		:= FALSE;
xCombiSynchroInProgress	:= FALSE;

xEncEmulationEnable	:= FALSE;
END_ACTION
TRANSITION FROM CombiExit TO ModeSelection:=
xExitStep
END_TRANSITION
(* @SFCISJUMP := 'ModeSelection' *)
TRANSITION FROM ModeSelection TO Posit:=
xPositioningMode
END_TRANSITION
STEP Posit:
IF (*NOT xInputPositioning*) xPositioningDone OR xReactionActive THEN
	xPositioningMode	:=	FALSE;
END_IF

xPositioningActive	:= TRUE;

CASE uiPositioningStep OF
	0:
		IF	VAR_Machine.iq_stParameter.i_uiAxisSelected >= CST_FillerSubModuleHmiStart AND
			VAR_Machine.iq_stParameter.i_uiAxisSelected <= CST_FillerSubModuleHmiStart + CST_LastFillerModuleAxis	THEN

			VAR_Machine.stFillerModule.iq_stParameters.i_uiAxisSelected
				:=	VAR_Machine.iq_stParameter.i_uiAxisSelected - CST_FillerSubModuleHmiStart;

			VAR_Machine.stFillerModule.iq_stParameters.i_rPositioningOffset
				:=	LREAL_TO_REAL(FC_TeensOfmmToDegrees(VAR_Machine.iq_stParameter.i_uiPositioningOffset, CFG_MC.Mechanical.MachineStep, FALSE, FALSE));

			uiPositioningStep	:=	100;
		ELSIF VAR_Machine.iq_stParameter.i_uiAxisSelected >= CST_InletSubModuleHmiStart AND
			VAR_Machine.iq_stParameter.i_uiAxisSelected <= CST_InletSubModuleHmiStart + CST_LastInletModuleAxis THEN

			VAR_Machine.stInletModule.iq_stParameters.i_uiAxisSelected
				:=	VAR_Machine.iq_stParameter.i_uiAxisSelected - CST_InletSubModuleHmiStart;

			VAR_Machine.stInletModule.iq_stParameters.i_rPositioningOffset
				:=	LREAL_TO_REAL(FC_TeensOfmmToDegrees(VAR_Machine.iq_stParameter.i_uiPositioningOffset, CFG_MC.Mechanical.MachineStep, FALSE, FALSE));

			uiPositioningStep	:=	200;
		ELSIF 	VAR_Machine.iq_stParameter.i_uiAxisSelected >= CST_OutletSubModuleHmiStart AND
			VAR_Machine.iq_stParameter.i_uiAxisSelected <= CST_OutletSubModuleHmiStart + CST_LastOutletModuleAxis THEN

			VAR_Machine.stOutletModule.iq_stParameters.i_uiAxisSelected
				:=	VAR_Machine.iq_stParameter.i_uiAxisSelected - CST_OutletSubModuleHmiStart;

			VAR_Machine.stOutletModule.iq_stParameters.i_rPositioningOffset
				:=	LREAL_TO_REAL(FC_TeensOfmmToDegrees(VAR_Machine.iq_stParameter.i_uiPositioningOffset, CFG_MC.Mechanical.MachineStep, FALSE, FALSE));

			uiPositioningStep	:=	300;
		ELSIF VAR_Machine.iq_stParameter.i_uiAxisSelected = CST_MachinePhasingOffset THEN
			uiPositioningStep	:=	700;
		END_IF

	100:(* Positioning On Filler Module *)
		VAR_Machine.stFillerModule.iq_stCmd.i_xPositioningMode :=	TRUE;

		IF VAR_Machine.stFillerModule.iq_stStatus.q_xPositioningActive 	AND
			VAR_Machine.stFillerModule.iq_stStatus.q_xPositioningDone	THEN

			VAR_Machine.stFillerModule.iq_stCmd.i_xPositioningMode 			:=	FALSE;
			VAR_Machine.stFillerModule.iq_stParameters.i_rPositioningOffset	:=	0.0;
			VAR_Machine.stFillerModule.iq_stParameters.i_uiAxisSelected		:=	CST_FirstFillerModuleAxis;
			uiPositioningStep	:=	150;
		END_IF

	150:
		IF NOT VAR_Machine.stFillerModule.iq_stStatus.q_xPositioningActive 	AND
			NOT VAR_Machine.stFillerModule.iq_stStatus.q_xPositioningDone	THEN
			uiPositioningStep	:=	400;
		END_IF

	200:(* Positioning On Inlet Module *)
		VAR_Machine.stInletModule.iq_stCmd.i_xPositioningMode :=	TRUE;

		IF VAR_Machine.stInletModule.iq_stStatus.q_xPositioningActive	AND
			VAR_Machine.stInletModule.iq_stStatus.q_xPositioningDone	THEN

			VAR_Machine.stInletModule.iq_stCmd.i_xPositioningMode 			:=	FALSE;
			VAR_Machine.stInletModule.iq_stParameters.i_rPositioningOffset	:=	0.0;
			VAR_Machine.stInletModule.iq_stParameters.i_uiAxisSelected		:=	CST_FirstInletModuleAxis;
			uiPositioningStep	:=	250;
		END_IF

	250:
		IF NOT VAR_Machine.stInletModule.iq_stStatus.q_xPositioningActive 	AND
			NOT	VAR_Machine.stInletModule.iq_stStatus.q_xPositioningDone	THEN
			uiPositioningStep	:=	400;
		END_IF

	300:(* Positioning On Outlet Module *)
		VAR_Machine.stOutletModule.iq_stCmd.i_xPositioningMode :=	TRUE;

		IF VAR_Machine.stOutletModule.iq_stStatus.q_xPositioningActive	AND
			VAR_Machine.stOutletModule.iq_stStatus.q_xPositioningDone	THEN

			VAR_Machine.stOutletModule.iq_stCmd.i_xPositioningMode 			:=	FALSE;
			VAR_Machine.stOutletModule.iq_stParameters.i_rPositioningOffset	:=	0.0;
			VAR_Machine.stOutletModule.iq_stParameters.i_uiAxisSelected		:=	CST_FirstOutletModuleAxis;
			uiPositioningStep	:=	350;
		END_IF

	350:
		IF NOT VAR_Machine.stOutletModule.iq_stStatus.q_xPositioningActive	AND
			NOT	VAR_Machine.stOutletModule.iq_stStatus.q_xPositioningDone	THEN
			uiPositioningStep	:=	400;
		END_IF

	400:
		xPositioningDone := TRUE;

	700:
		VAR_Machine.stFillerModule.iq_stCmd.i_xAutoMode	:=	TRUE;
		VAR_Machine.stOutletModule.iq_stCmd.i_xAutoMode	:=	VAR_Machine.stOutletModule.iq_stStatus.q_xModuleReal;
		VAR_Machine.stInletModule.iq_stCmd.i_xAutoMode	:=	VAR_Machine.stInletModule.iq_stStatus.q_xModuleReal;

		uiPositioningStep	:=	710;

	710:(* The machine is rephased *)
		IF VAR_Machine.stFillerModule.iq_stStatus.q_xAutoActive		AND
			(VAR_Machine.stInletModule.iq_stStatus.q_xAutoActive	OR NOT
			VAR_Machine.stInletModule.iq_stStatus.q_xModuleReal)	AND
			(VAR_Machine.stOutletModule.iq_stStatus.q_xAutoActive	OR NOT
			VAR_Machine.stOutletModule.iq_stStatus.q_xModuleReal)	THEN

			IF 	NOT VAR_Machine.stFillerModule.iq_stStatus.q_xSynchroWithOffset	AND
				NOT VAR_Machine.stInletModule.iq_stStatus.q_xSynchroWithOffset	AND
				NOT VAR_Machine.stOutletModule.iq_stStatus.q_xSynchroWithOffset	THEN

				VAR_Machine.stMasterModule.iq_stParameters.i_lrRephasingPosition	:=
					FC_RephasingMachine(iq_astInletSubModuleAxis	:=	VAR_Machine.stInletModule.iq_astSubModuleAxis,
										iq_astFillerSubModuleAxis	:=	VAR_Machine.stFillerModule.iq_astSubModuleAxis,
										iq_astOutletSubModuleAxis	:=	VAR_Machine.stOutletModule.iq_astSubModuleAxis);

				VAR_Machine.stFillerModule.iq_stParameters.i_lrRephasingPosition	:=	VAR_Machine.stMasterModule.iq_stParameters.i_lrRephasingPosition;
				VAR_Machine.stOutletModule.iq_stParameters.i_lrRephasingPosition	:=	VAR_Machine.stMasterModule.iq_stParameters.i_lrRephasingPosition;
				VAR_Machine.stInletModule.iq_stParameters.i_lrRephasingPosition		:=	VAR_Machine.stMasterModule.iq_stParameters.i_lrRephasingPosition;

				uiPositioningStep	:=	740;
			END_IF
		END_IF

	740:
		VAR_Machine.stMasterModule.iq_stCmd.i_xPositioning				:=	TRUE;
		VAR_Machine.stMasterModule.iq_stCmd.i_xMasterRephasingRequest	:= 	TRUE;

		IF VAR_Machine.stMasterModule.iq_stStatus.q_xPositioningActive AND VAR_Machine.stMasterModule.iq_stStatus.q_xMasterRephased THEN
			VAR_Machine.stMasterModule.iq_stCmd.i_xMasterRephasingRequest	:= 	FALSE;
			uiPositioningStep	:=	750;
		END_IF

	750:
		VAR_Machine.stFillerModule.iq_stCmd.i_xStart	:=	TRUE;
		VAR_Machine.stInletModule.iq_stCmd.i_xStart		:=	VAR_Machine.stInletModule.iq_stStatus.q_xModuleReal;
		VAR_Machine.stOutletModule.iq_stCmd.i_xStart	:=	VAR_Machine.stOutletModule.iq_stStatus.q_xModuleReal;
		uiPositioningStep	:=	760;

	760:
		IF VAR_Machine.stFillerModule.iq_stStatus.q_xRealAxesSynchronized		AND
			VAR_Machine.stFillerModule.iq_stStatus.q_xAutoActive				AND
			VAR_Machine.stFillerModule.iq_stStatus.q_xMasterRephased			AND

			((VAR_Machine.stInletModule.iq_stStatus.q_xRealAxesSynchronized		AND
			VAR_Machine.stInletModule.iq_stStatus.q_xMasterRephased				AND
			VAR_Machine.stInletModule.iq_stStatus.q_xAutoActive)				OR NOT
			VAR_Machine.stInletModule.iq_stStatus.q_xModuleReal)				AND

			((VAR_Machine.stOutletModule.iq_stStatus.q_xRealAxesSynchronized	AND
			VAR_Machine.stOutletModule.iq_stStatus.q_xMasterRephased			AND
			VAR_Machine.stOutletModule.iq_stStatus.q_xAutoActive)				OR NOT
			VAR_Machine.stOutletModule.iq_stStatus.q_xModuleReal)				THEN

			VAR_Machine.stMasterModule.iq_stParameters.i_rPositioningOffset	:= LREAL_TO_REAL(FC_TeensOfmmToDegrees(VAR_Machine.iq_stParameter.i_uiPositioningOffset, CFG_MC.Mechanical.MachineStep, FALSE, TRUE));
			VAR_Machine.stMasterModule.iq_stCmd.i_xStart	:=	TRUE;
			uiPositioningStep	:=	770;
		END_IF

	770:
		IF VAR_Machine.stMasterModule.iq_stStatus.q_xPositioningDone THEN
			VAR_Machine.stMasterModule.iq_stCmd.i_xStart		:= FALSE;
			uiPositioningStep	:=	780;	//v1.2
		END_IF

	780:	//v1.2
		IF VAR_Machine.stMasterModule.iq_stStatus.q_xModuleStopped THEN	//v1.2
			VAR_Machine.stFillerModule.iq_stCmd.i_xStart	:= FALSE;	//v1.2
			VAR_Machine.stInletModule.iq_stCmd.i_xStart		:= FALSE;	//v1.2
			VAR_Machine.stOutletModule.iq_stCmd.i_xStart	:= FALSE;	//v1.2
			VAR_Machine.stFillerModule.iq_stCmd.i_xAutoMode	:= FALSE;	//v1.2
			VAR_Machine.stInletModule.iq_stCmd.i_xAutoMode	:= FALSE;	//v1.2
			VAR_Machine.stOutletModule.iq_stCmd.i_xAutoMode	:= FALSE;	//v1.2
			uiPositioningStep	:=	790;	//v1.2
		END_IF	//v1.2

	790:	//v1.2
		IF NOT VAR_Machine.stFillerModule.iq_stStatus.q_xAutoActive AND	//v1.2
			NOT VAR_Machine.stInletModule.iq_stStatus.q_xAutoActive AND	//v1.2
			NOT VAR_Machine.stOutletModule.iq_stStatus.q_xAutoActive THEN	//v1.2

			uiPositioningStep	:=	800;	//v1.2
		END_IF	//v1.2

	800:	//v1.2
		VAR_Machine.stMasterModule.iq_stCmd.i_xPositioning	:= FALSE;	//v1.2
		xPositioningDone := TRUE;	//v1.2
END_CASE
END_STEP
ENTRY_ACTION
uiPositioningStep	:=	0;
xPositioningDone	:=	FALSE;
END_ACTION
EXIT_ACTION
VAR_Machine.stFillerModule.iq_stCmd.i_xPositioningMode 			:= FALSE;
VAR_Machine.stFillerModule.iq_stCmd.i_xStart					:= FALSE;	//v1.2
VAR_Machine.stFillerModule.iq_stParameters.i_rPositioningOffset	:= 0.0;
VAR_Machine.stFillerModule.iq_stParameters.i_uiAxisSelected		:= CST_FirstFillerModuleAxis;
VAR_Machine.stFillerModule.iq_stCmd.i_xAutoMode					:= FALSE;

VAR_Machine.stOutletModule.iq_stCmd.i_xPositioningMode			:= FALSE;
VAR_Machine.stOutletModule.iq_stCmd.i_xStart					:= FALSE;	//v1.2
VAR_Machine.stOutletModule.iq_stParameters.i_rPositioningOffset	:= 0.0;
VAR_Machine.stOutletModule.iq_stParameters.i_uiAxisSelected		:= CST_FirstOutletModuleAxis;
VAR_Machine.stOutletModule.iq_stCmd.i_xAutoMode					:= FALSE;

VAR_Machine.stInletModule.iq_stCmd.i_xPositioningMode			:= FALSE;
VAR_Machine.stInletModule.iq_stCmd.i_xStart						:= FALSE;	//v1.2
VAR_Machine.stInletModule.iq_stParameters.i_rPositioningOffset	:= 0.0;
VAR_Machine.stInletModule.iq_stParameters.i_uiAxisSelected		:= CST_FirstInletModuleAxis;
VAR_Machine.stInletModule.iq_stCmd.i_xAutoMode					:= FALSE;
END_ACTION
TRANSITION FROM Posit TO PositExit:=
NOT xPositioningMode
END_TRANSITION
STEP PositExit:
xExitStep			:= 	TRUE;
xPositioningDone	:=	FALSE;
xPositioningActive	:=	FALSE;
END_STEP
TRANSITION FROM PositExit TO ModeSelection:=
xExitStep
END_TRANSITION
(* @SFCISJUMP := 'ModeSelection' *)
TRANSITION FROM ModeSelection TO Velocity:=
xVelocityMode
END_TRANSITION
STEP Velocity:
IF NOT xInputVelocity OR xReactionActive THEN
	xVelocityMode	:= FALSE;
END_IF

xVelocityActive	:= TRUE;

CASE uiVelocityStep OF
	0:
		IF VAR_Machine.iq_stParameter.i_uiAxisSelected >= CST_FillerSubModuleHmiStart AND
			VAR_Machine.iq_stParameter.i_uiAxisSelected <= CST_FillerSubModuleHmiStart + CST_LastFillerModuleAxis	THEN

			VAR_Machine.stFillerModule.iq_stParameters.i_uiAxisSelected	:= VAR_Machine.iq_stParameter.i_uiAxisSelected - CST_FillerSubModuleHmiStart;
			uiVelocityStep	:= 100;
		ELSIF VAR_Machine.iq_stParameter.i_uiAxisSelected >= CST_InletSubModuleHmiStart AND
			VAR_Machine.iq_stParameter.i_uiAxisSelected <= CST_InletSubModuleHmiStart + CST_LastInletModuleAxis THEN

			VAR_Machine.stInletModule.iq_stParameters.i_uiAxisSelected	:= VAR_Machine.iq_stParameter.i_uiAxisSelected - CST_InletSubModuleHmiStart;
			uiVelocityStep	:= 200;
		ELSIF VAR_Machine.iq_stParameter.i_uiAxisSelected >= CST_OutletSubModuleHmiStart AND
			VAR_Machine.iq_stParameter.i_uiAxisSelected <= CST_OutletSubModuleHmiStart + CST_LastOutletModuleAxis THEN

			VAR_Machine.stOutletModule.iq_stParameters.i_uiAxisSelected	:= VAR_Machine.iq_stParameter.i_uiAxisSelected - CST_OutletSubModuleHmiStart;
			uiVelocityStep	:= 300;
		END_IF

	100:(* Velocity On Filler Module *)
		VAR_Machine.stFillerModule.iq_stCmd.i_xVelocityMode 			:= TRUE;
		VAR_Machine.stFillerModule.iq_stParameters.i_rManualVelocity	:= UINT_TO_REAL(VAR_Machine.iq_stParameter.i_uiManualVelocity);

		IF 	VAR_Machine.stFillerModule.iq_stStatus.q_xVelocityActive THEN
			VAR_Machine.stFillerModule.iq_stCmd.i_xStart	:= TRUE;
		END_IF

	200:(* Velocity On Inlet Module *)
		VAR_Machine.stInletModule.iq_stCmd.i_xVelocityMode 			:= TRUE;
		VAR_Machine.stInletModule.iq_stParameters.i_rManualVelocity	:= UINT_TO_REAL(VAR_Machine.iq_stParameter.i_uiManualVelocity);

		IF 	VAR_Machine.stInletModule.iq_stStatus.q_xVelocityActive THEN
			VAR_Machine.stInletModule.iq_stCmd.i_xStart	:= TRUE;
		END_IF

	300:(* Velocity On Outlet Module *)
		VAR_Machine.stOutletModule.iq_stCmd.i_xVelocityMode 			:= TRUE;
		VAR_Machine.stOutletModule.iq_stParameters.i_rManualVelocity	:= UINT_TO_REAL(VAR_Machine.iq_stParameter.i_uiManualVelocity);

		IF 	VAR_Machine.stOutletModule.iq_stStatus.q_xVelocityActive THEN
			VAR_Machine.stOutletModule.iq_stCmd.i_xStart	:= TRUE;
		END_IF
END_CASE
END_STEP
ENTRY_ACTION
uiVelocityStep	:=	0;
END_ACTION
EXIT_ACTION
VAR_Machine.stFillerModule.iq_stCmd.i_xStart		:=	FALSE;
VAR_Machine.stFillerModule.iq_stCmd.i_xVelocityMode :=	FALSE;

VAR_Machine.stOutletModule.iq_stCmd.i_xStart		:=	FALSE;
VAR_Machine.stOutletModule.iq_stCmd.i_xVelocityMode :=	FALSE;

VAR_Machine.stInletModule.iq_stCmd.i_xStart			:=	FALSE;
VAR_Machine.stInletModule.iq_stCmd.i_xVelocityMode :=	FALSE;

xVelocityActive	:=	FALSE;
END_ACTION
TRANSITION FROM Velocity TO VelExit:=
NOT xVelocityMode
END_TRANSITION
STEP VelExit:
xExitStep	:= VAR_Machine.iq_stStatus.q_xMachineStopped;
END_STEP
TRANSITION FROM VelExit TO Init:=
xExitStep
END_TRANSITION
(* @SFCISJUMP := 'Init' *)
TRANSITION FROM ModeSelection TO SelectiveHome:=
xSelectiveHomingMode
END_TRANSITION
STEP SelectiveHome:
IF xReactionActive  OR NOT xInputSelHoming THEN
	xSelectiveHomingMode	:=	FALSE;
END_IF

xSelHomingActive	:= TRUE;

CASE uiSelectiveHomingStep OF
	0:
		IF VAR_Machine.iq_stParameter.i_uiAxisSelected >= CST_FillerSubModuleHmiStart AND
			VAR_Machine.iq_stParameter.i_uiAxisSelected <= CST_FillerSubModuleHmiStart + CST_LastFillerModuleAxis	THEN

			VAR_Machine.stFillerModule.iq_stParameters.i_uiAxisSelected	:=	VAR_Machine.iq_stParameter.i_uiAxisSelected - CST_FillerSubModuleHmiStart;
			uiSelectiveHomingStep	:=	100;
		ELSIF VAR_Machine.iq_stParameter.i_uiAxisSelected >= CST_OutletSubModuleHmiStart AND
			VAR_Machine.iq_stParameter.i_uiAxisSelected <= CST_OutletSubModuleHmiStart + CST_LastOutletModuleAxis THEN

			VAR_Machine.stOutletModule.iq_stParameters.i_uiAxisSelected	:=	VAR_Machine.iq_stParameter.i_uiAxisSelected - CST_OutletSubModuleHmiStart;
			uiSelectiveHomingStep	:=	200;
		ELSIF VAR_Machine.iq_stParameter.i_uiAxisSelected >= CST_InletSubModuleHmiStart AND
			VAR_Machine.iq_stParameter.i_uiAxisSelected <= CST_InletSubModuleHmiStart + CST_LastInletModuleAxis THEN

			VAR_Machine.stInletModule.iq_stParameters.i_uiAxisSelected	:=	VAR_Machine.iq_stParameter.i_uiAxisSelected - CST_InletSubModuleHmiStart;
			uiSelectiveHomingStep	:=	300;
		ELSIF VAR_Machine.iq_stParameter.i_uiAxisSelected =	CST_MachinePhasingOffset THEN
			uiSelectiveHomingStep	:=	800;
		END_IF

	100:(* Homing On Filler Module *)
		VAR_Machine.stFillerModule.iq_stCmd.i_xSelectiveHomingMode :=	TRUE;

		IF VAR_Machine.stFillerModule.iq_stStatus.q_xSelHomingActive AND VAR_Machine.stFillerModule.iq_stStatus.q_xSelHomingDone THEN
			VAR_Machine.stFillerModule.iq_stCmd.i_xSelectiveHomingMode 		:=	FALSE;
			VAR_Machine.stFillerModule.iq_stParameters.i_uiAxisSelected		:=	CST_FirstFillerModuleAxis;
			uiSelectiveHomingStep	:=	150;
		END_IF

	150:
		IF NOT VAR_Machine.stFillerModule.iq_stStatus.q_xSelHomingActive AND NOT VAR_Machine.stFillerModule.iq_stStatus.q_xSelHomingDone THEN
			uiSelectiveHomingStep	:=	400;
		END_IF

	200:(* Homing On Outlet Module *)
		VAR_Machine.stOutletModule.iq_stCmd.i_xSelectiveHomingMode :=	TRUE;

		IF VAR_Machine.stOutletModule.iq_stStatus.q_xSelHomingActive AND VAR_Machine.stOutletModule.iq_stStatus.q_xSelHomingDone THEN
			VAR_Machine.stOutletModule.iq_stCmd.i_xSelectiveHomingMode 		:=	FALSE;
			VAR_Machine.stOutletModule.iq_stParameters.i_uiAxisSelected		:=	CST_FirstOutletModuleAxis;
			uiSelectiveHomingStep	:=	250;
		END_IF

	250:
		IF NOT VAR_Machine.stOutletModule.iq_stStatus.q_xSelHomingActive AND NOT VAR_Machine.stOutletModule.iq_stStatus.q_xSelHomingDone THEN
			uiSelectiveHomingStep	:=	400;
		END_IF

	300:(* Homing On Inlet Module *)
		VAR_Machine.stInletModule.iq_stCmd.i_xSelectiveHomingMode :=	TRUE;

		IF VAR_Machine.stInletModule.iq_stStatus.q_xSelHomingActive AND VAR_Machine.stInletModule.iq_stStatus.q_xSelHomingDone THEN
			VAR_Machine.stInletModule.iq_stCmd.i_xSelectiveHomingMode 		:=	FALSE;
			VAR_Machine.stInletModule.iq_stParameters.i_uiAxisSelected		:=	CST_FirstInletModuleAxis;
			uiSelectiveHomingStep	:=	350;
		END_IF

	350:
		IF NOT VAR_Machine.stInletModule.iq_stStatus.q_xSelHomingActive AND NOT	VAR_Machine.stInletModule.iq_stStatus.q_xSelHomingDone THEN
			uiSelectiveHomingStep	:=	400;
		END_IF

	400:

	800:(* Homing On Master Module *)
		VAR_Machine.stMasterModule.iq_stCmd.i_xSelectiveHomingMode :=	TRUE;

		IF VAR_Machine.stMasterModule.iq_stStatus.q_xSelHomingActive AND VAR_Machine.stMasterModule.iq_stStatus.q_xSelHomingDone THEN
			VAR_Machine.stMasterModule.iq_stCmd.i_xSelectiveHomingMode 		:=	FALSE;
			VAR_Machine.stMasterModule.iq_stParameters.i_uiAxisSelected		:=	CST_MachinePhasingOffset;
			uiSelectiveHomingStep	:=	850;
		END_IF

	850:
		IF NOT VAR_Machine.stMasterModule.iq_stStatus.q_xSelHomingActive AND NOT	VAR_Machine.stMasterModule.iq_stStatus.q_xSelHomingDone THEN
			uiSelectiveHomingStep	:=	400;
		END_IF
END_CASE
END_STEP
ENTRY_ACTION
uiSelectiveHomingStep	:=	0;
END_ACTION
EXIT_ACTION
VAR_Machine.stFillerModule.iq_stCmd.i_xSelectiveHomingMode 		:=	FALSE;
VAR_Machine.stFillerModule.iq_stParameters.i_uiAxisSelected		:=	CST_FirstFillerModuleAxis;

VAR_Machine.stInletModule.iq_stCmd.i_xSelectiveHomingMode		:=	FALSE;
VAR_Machine.stInletModule.iq_stParameters.i_uiAxisSelected		:=	CST_FirstInletModuleAxis;

VAR_Machine.stOutletModule.iq_stCmd.i_xSelectiveHomingMode		:=	FALSE;
VAR_Machine.stOutletModule.iq_stParameters.i_uiAxisSelected		:=	CST_FirstOutletModuleAxis;

VAR_Machine.stMasterModule.iq_stCmd.i_xSelectiveHomingMode		:=	FALSE;
VAR_Machine.stMasterModule.iq_stParameters.i_uiAxisSelected		:=	CST_MachinePhasingOffset;
END_ACTION
TRANSITION FROM SelectiveHome TO SelHomeExit:=
NOT xSelectiveHomingMode
END_TRANSITION
STEP SelHomeExit:
xExitStep	:= TRUE;
END_STEP
TRANSITION FROM SelHomeExit TO ModeSelection:=
xExitStep
END_TRANSITION
(* @SFCISJUMP := 'ModeSelection' *)
TRANSITION FROM ModeSelection TO Multi:=
xMultiMode
END_TRANSITION
STEP Multi:
IF NOT xInputMulti	THEN
	VAR_Machine.stOutletModule.iq_stCmd.i_xStart					:= FALSE;
	VAR_Machine.stOutletModule.iq_stCmd.i_xAutoMultiMode			:= FALSE;
	VAR_Machine.stOutletModule.iq_stCmd.i_xJogMultiMode				:= FALSE;
	VAR_Machine.stOutletModule.iq_stCmd.i_xJogPB					:= FALSE;

	VAR_Machine.stInletModule.iq_stCmd.i_xStart						:= FALSE;
	VAR_Machine.stInletModule.iq_stCmd.i_xAutoMultiMode				:= FALSE;
	VAR_Machine.stInletModule.iq_stCmd.i_xJogMultiMode				:= FALSE;
	VAR_Machine.stInletModule.iq_stCmd.i_xJogPB						:= FALSE;

	VAR_Machine.stFillerModule.iq_stCmd.i_xStart					:= FALSE;
	VAR_Machine.stFillerModule.iq_stCmd.i_xAutoMultiMode			:= FALSE;
	VAR_Machine.stFillerModule.iq_stCmd.i_xJogMultiMode				:= FALSE;
	VAR_Machine.stFillerModule.iq_stCmd.i_xJogPB					:= FALSE;

	VAR_Machine.stInletModule.iq_stCmd.i_xSlowMotionForward			:= FALSE;
	VAR_Machine.stInletModule.iq_stCmd.i_xSlowMotionBackward		:= FALSE;

	VAR_Machine.stOutletModule.iq_stCmd.i_xSlowMotionForward		:= FALSE;
	VAR_Machine.stOutletModule.iq_stCmd.i_xSlowMotionBackward		:= FALSE;

	IF VAR_Machine.stFillerModule.iq_stStatus.q_xModuleStopped		AND
		(VAR_Machine.stInletModule.iq_stStatus.q_xModuleStopped		OR NOT VAR_Machine.stInletModule.iq_stStatus.q_xModuleReal)		AND
		(VAR_Machine.stOutletModule.iq_stStatus.q_xModuleStopped	OR NOT VAR_Machine.stOutletModule.iq_stStatus.q_xModuleReal)	THEN
		xMultiMode	:= FALSE;
	END_IF
END_IF

xMultiActive	:= TRUE;

xReactionOnFillerModule		:= xReactFillerEmergencyStop 	OR xReactFillerQuickStop		OR xReactFillerStop	OR NOT xInputMulti	OR
								(uiFillerMultiStep >= 100	AND  uiFillerMultiStep < 200 	AND NOT MC_InputOutput.Network.Filler.Commands.JogFillerModule) OR
								(uiFillerMultiStep >= 500	AND  uiFillerMultiStep < 900 	AND NOT MC_InputOutput.Network.Filler.Commands.AutoFillerModule);

IF xReactionOnFillerModule THEN
	IF uiFillerMultiStep <> 1000 AND uiFillerMultiStep <> 0 THEN
		uiFillerMultiStep	:=	1000;
	END_IF
END_IF

CASE uiFillerMultiStep OF
	0:(* Modality selecetion *)
		IF NOT xReactionOnFillerModule THEN
			IF MC_InputOutput.Network.Filler.Commands.JogFillerModule THEN
				uiFillerMultiStep	:=	100;
			ELSIF MC_InputOutput.Network.Filler.Commands.AutoFillerModule THEN
				uiFillerMultiStep	:=	500;
			END_IF
		END_IF

	100:(* Jog Multy *)
		VAR_Machine.stFillerModule.iq_stCmd.i_xJogMultiMode := TRUE;
		uiFillerMultiStep := 110;

	110:(* Wait for jog active on filler module and axes without offset *)
		IF VAR_Machine.stFillerModule.iq_stStatus.q_xJogMultiActive THEN
			IF NOT VAR_Machine.stFillerModule.iq_stStatus.q_xSynchroWithOffset THEN
				VAR_Machine.stFillerModule.iq_stCmd.i_xMasterRephasingRequest		:= TRUE;
				VAR_Machine.stFillerModule.iq_stParameters.i_lrRephasingPosition	:= FC_RephasingPositionFiller(iq_astSubModuleAxis := VAR_Machine.stFillerModule.iq_astSubModuleAxis);
				VAR_Machine.iq_stCmd.i_xStart										:= TRUE;
				uiFillerMultiStep := 120;
			END_IF
		END_IF

	120:(* Rephasing of master position *)
		IF  VAR_Machine.stFillerModule.iq_stStatus.q_xMasterRephased THEN
			VAR_Machine.stFillerModule.iq_stCmd.i_xMasterRephasingRequest	:= 	FALSE;
			uiFillerMultiStep := 130;
		END_IF

	130:(* Jog Push button *)
		VAR_Machine.stFillerModule.iq_stCmd.i_xJogPB :=	MC_InputOutput.Network.Filler.Commands.JogPushButtonFillerModule;
		IF VAR_Machine.stFillerModule.iq_stCmd.i_xJogPB THEN
			uiFillerMultiStep := 140;
		END_IF

	140:
		VAR_Machine.stFillerModule.iq_stCmd.i_xJogPB := MC_InputOutput.Network.Filler.Commands.JogPushButtonFillerModule;
		IF NOT VAR_Machine.stFillerModule.iq_stCmd.i_xJogPB THEN
			VAR_Machine.stFillerModule.iq_stCmd.i_xJogMultiMode	:= FALSE;
			uiFillerMultiStep := 160;
		END_IF

	160:
		IF VAR_Machine.stFillerModule.iq_stStatus.q_xModuleStopped AND NOT VAR_Machine.stFillerModule.iq_stStatus.q_xJogMultiActive	THEN
			uiFillerMultiStep := 100;
		END_IF

	500:
		VAR_Machine.stFillerModule.iq_stCmd.i_xAutoMultiMode := TRUE;
		uiFillerMultiStep := 510;

	510:(* The phase compensation process has to be ended bofore going on next steps *)
		IF VAR_Machine.stFillerModule.iq_stStatus.q_xAutoMultiActive THEN
			IF NOT VAR_Machine.stFillerModule.iq_stStatus.q_xSynchroWithOffset THEN
				VAR_Machine.stFillerModule.iq_stParameters.i_lrRephasingPosition	:= FC_RephasingPositionFiller(iq_astSubModuleAxis := VAR_Machine.stFillerModule.iq_astSubModuleAxis);
				uiFillerMultiStep := 520;
			END_IF
		END_IF

	520:(* Rephasing position of the master *)
		VAR_Machine.stFillerModule.iq_stCmd.i_xMasterRephasingRequest	:= TRUE;
		uiFillerMultiStep := 525;//V4.A.A.1.6.12d

	525://V4.A.A.1.6.12d
		IF VAR_Machine.stFillerModule.iq_stStatus.q_xMasterRephased THEN
			VAR_Machine.stFillerModule.iq_stCmd.i_xMasterRephasingRequest	:= 	FALSE;
			uiFillerMultiStep := 530;
		END_IF

	530:(* Wait the start command from the plc *)
		IF MC_InputOutput.Network.Filler.Commands.StartFillerModule THEN
			VAR_Machine.stFillerModule.iq_stCmd.i_xStart := TRUE;
			uiFillerMultiStep := 540;
		END_IF

	540:
		IF NOT MC_InputOutput.Network.Filler.Commands.StartFillerModule THEN
			VAR_Machine.stFillerModule.iq_stCmd.i_xStart := FALSE;
			uiFillerMultiStep	:= 545;
		ELSIF VAR_Machine.iq_stCmd.i_xAxisPhaseShift THEN
			IF VAR_Machine.iq_stParameter.i_uiAxisSelected >= CST_FillerSubModuleHmiStart AND
				VAR_Machine.iq_stParameter.i_uiAxisSelected <= CST_FillerSubModuleHmiStart + CST_LastFillerModuleAxis THEN

				VAR_Machine.stFillerModule.iq_stParameters.i_uiAxisSelected			:= VAR_Machine.iq_stParameter.i_uiAxisSelected - CST_FillerSubModuleHmiStart;
				VAR_Machine.stFillerModule.iq_stParameters.i_rPhaseShiftDistance	:= LREAL_TO_REAL(FC_TeensOfmmToDegrees(VAR_Machine.iq_stParameter.i_iAxisPhaseShiftDistance, CFG_MC.Mechanical.MachineStep, TRUE, FALSE));

				uiFillerMultiStep	:=	600;
			END_IF
		END_IF

	545:
		IF VAR_Machine.stFillerModule.iq_stStatus.q_xModuleStopped THEN
			uiFillerMultiStep	:=	550;
		END_IF

	550:
		IF MC_InputOutput.Network.Filler.Commands.StartFillerModule THEN
			VAR_Machine.stFillerModule.iq_stCmd.i_xStart	:= TRUE;
			uiFillerMultiStep	:=	540;
		ELSIF VAR_Machine.stMasterModule.iq_stStatus.q_xSynchroWithOffset OR VAR_Machine.stFillerModule.iq_stStatus.q_xSynchroWithOffset	THEN
			uiFillerMultiStep	:= 800;
		END_IF

	600:
		VAR_Machine.stFillerModule.iq_stCmd.i_xPhaseShift := TRUE;
		uiFillerMultiStep	:= 610;

	610:
		IF VAR_Machine.stFillerModule.iq_stStatus.q_xPhaseShiftDone AND NOT VAR_Machine.iq_stCmd.i_xAxisPhaseShift THEN
			VAR_Machine.stFillerModule.iq_stCmd.i_xPhaseShift	:= FALSE;
			uiFillerMultiStep	:= 540;
		END_IF

	800:
		VAR_Machine.stFillerModule.iq_stCmd.i_xPhaseCompensation := VAR_Machine.stFillerModule.iq_stStatus.q_xSynchroWithOffset;
		uiFillerMultiStep	:= 810;

	810:
		IF NOT VAR_Machine.stFillerModule.iq_stStatus.q_xSynchroWithOffset	THEN
			VAR_Machine.stFillerModule.iq_stCmd.i_xPhaseCompensation	:= FALSE;
			uiFillerMultiStep	:= 550;
		END_IF

	1000:
		IF VAR_Machine.stFillerModule.iq_stStatus.q_xModuleStopped THEN
			VAR_Machine.stFillerModule.iq_stCmd.i_xJogMultiMode		:= FALSE;
			VAR_Machine.stFillerModule.iq_stCmd.i_xAutoMultiMode	:= FALSE;
			uiFillerMultiStep	:=	0;
		END_IF

		VAR_Machine.stFillerModule.iq_stCmd.i_xJogPB					:= FALSE;
		VAR_Machine.stFillerModule.iq_stCmd.i_xPhaseShift				:= FALSE;
		VAR_Machine.stFillerModule.iq_stCmd.i_xStart					:= FALSE;
		VAR_Machine.stFillerModule.iq_stCmd.i_xAutoMultiMode			:= FALSE;
		VAR_Machine.stFillerModule.iq_stCmd.i_xJogMultiMode				:= FALSE;
		VAR_Machine.stFillerModule.iq_stCmd.i_xMasterRephasingRequest	:= FALSE;
		VAR_Machine.stFillerModule.iq_stCmd.i_xPhaseCompensation		:= FALSE;
END_CASE

xReactionOnInletModule	:= xReactInletEmergencyStop		OR xReactInletQuickStop 	OR xReactInletStop	OR NOT xInputMulti	OR
							(uiInletMultiStep >= 100	AND uiInletMultiStep < 200 	AND NOT MC_InputOutput.Network.Inlet.Commands.JogInletModule) 	OR
							(uiInletMultiStep >= 200	AND uiInletMultiStep < 500 	AND NOT xSlowMotionCommandInlet)		OR
							(uiInletMultiStep >= 500	AND uiInletMultiStep < 900 	AND NOT MC_InputOutput.Network.Inlet.Commands.AutoInletModule);

IF xReactionOnInletModule THEN
	IF uiInletMultiStep <> 1000 AND uiInletMultiStep <> 0 THEN
		uiInletMultiStep	:=	1000;
	END_IF
END_IF

CASE uiInletMultiStep OF
	0:(* Modality selecetion *)
		IF NOT xReactionOnInletModule THEN
			IF MC_InputOutput.Network.Inlet.Commands.JogInletModule AND NOT xSlowMotionCommandInlet THEN
				uiInletMultiStep	:=	100;
			ELSIF NOT MC_InputOutput.Network.Inlet.Commands.JogInletModule AND xSlowMotionCommandInlet THEN
				uiInletMultiStep	:=	200;
			ELSIF MC_InputOutput.Network.Inlet.Commands.AutoInletModule THEN
				uiInletMultiStep	:=	500;
			END_IF
		END_IF

	100:(* Jog Multy *)
		VAR_Machine.stInletModule.iq_stCmd.i_xJogMultiMode := TRUE;
		uiInletMultiStep := 110;

	110:(* Wait for jog active on Inlet module and axes without offset *)
		IF VAR_Machine.stInletModule.iq_stStatus.q_xJogMultiActive THEN
			IF NOT VAR_Machine.stInletModule.iq_stStatus.q_xSynchroWithOffset THEN
				VAR_Machine.stInletModule.iq_stCmd.i_xMasterRephasingRequest	:= TRUE;
				VAR_Machine.stInletModule.iq_stParameters.i_lrRephasingPosition	:= FC_RephasingPositionInlet(iq_astSubModuleAxis := VAR_Machine.stInletModule.iq_astSubModuleAxis);
				VAR_Machine.iq_stCmd.i_xStart									:= TRUE;
				uiInletMultiStep	:=	120;
			END_IF
		END_IF

	120:(* Rephasing of master position *)
		IF  VAR_Machine.stInletModule.iq_stStatus.q_xMasterRephased THEN
			VAR_Machine.stInletModule.iq_stCmd.i_xMasterRephasingRequest	:= 	FALSE;
			uiInletMultiStep	:=	130;
		END_IF

	130:(* Jog Push button *)
		VAR_Machine.stInletModule.iq_stCmd.i_xJogPB	:= MC_InputOutput.Network.Inlet.Commands.JogPushButtonInletModule;
		IF VAR_Machine.stInletModule.iq_stCmd.i_xJogPB THEN
			uiInletMultiStep	:=	140;
		END_IF

	140:
		VAR_Machine.stInletModule.iq_stCmd.i_xJogPB	:= MC_InputOutput.Network.Inlet.Commands.JogPushButtonInletModule;
		IF NOT VAR_Machine.stInletModule.iq_stCmd.i_xJogPB THEN
			VAR_Machine.stInletModule.iq_stCmd.i_xJogMultiMode	:= FALSE;
			uiInletMultiStep	:=	160;
		END_IF

	160:
		IF 	VAR_Machine.stInletModule.iq_stStatus.q_xModuleStopped AND NOT VAR_Machine.stInletModule.iq_stStatus.q_xJogMultiActive THEN
			uiInletMultiStep	:=	100;
		END_IF

	200:
		VAR_Machine.stInletModule.iq_stCmd.i_xSlowMotionForward		:= xSlowMotionCommandInletForward;
		VAR_Machine.stInletModule.iq_stCmd.i_xSlowMotionBackward	:= xSlowMotionCommandInletBackward;
		uiInletMultiStep	:=	230;

	230:
		IF VAR_Machine.stInletModule.iq_stStatus.q_xSlowMotionActive THEN
			uiInletMultiStep	:=	250;
		END_IF

	250:
		VAR_Machine.stInletModule.iq_stCmd.i_xSlowMotionForward		:= xSlowMotionCommandInletForward;
		VAR_Machine.stInletModule.iq_stCmd.i_xSlowMotionBackward	:= xSlowMotionCommandInletBackward;
		VAR_Machine.stInletModule.iq_stCmd.i_xJogPB					:= MC_InputOutput.Network.Inlet.Commands.JogPushButtonInletModule;

	500:
		VAR_Machine.stInletModule.iq_stCmd.i_xAutoMultiMode	:= TRUE;
		uiInletMultiStep	:=	510;

	510:(* The phase compensation process has to be ended bofore going on next steps *)
		IF VAR_Machine.stInletModule.iq_stStatus.q_xAutoMultiActive THEN
			IF NOT VAR_Machine.stInletModule.iq_stStatus.q_xSynchroWithOffset THEN
				VAR_Machine.stInletModule.iq_stParameters.i_lrRephasingPosition	:=	FC_RephasingPositionInlet(iq_astSubModuleAxis := VAR_Machine.stInletModule.iq_astSubModuleAxis);
				uiInletMultiStep	:=	520;
			END_IF
		END_IF

	520:(* Rephasing position of the master *)
		VAR_Machine.stInletModule.iq_stCmd.i_xMasterRephasingRequest	:= TRUE;

		IF  VAR_Machine.stInletModule.iq_stStatus.q_xMasterRephased THEN
			VAR_Machine.stInletModule.iq_stCmd.i_xMasterRephasingRequest	:= 	FALSE;
			uiInletMultiStep	:=	530;
		END_IF

	530:(* Wait the start command from the plc *)
		IF  MC_InputOutput.Network.Inlet.Commands.StartInletModule THEN
			VAR_Machine.stInletModule.iq_stCmd.i_xStart	:=	TRUE;
			uiInletMultiStep	:=	540;
		END_IF

	540:
		IF NOT MC_InputOutput.Network.Inlet.Commands.StartInletModule THEN
			VAR_Machine.stInletModule.iq_stCmd.i_xStart	:= FALSE;
			uiInletMultiStep	:= 545;
		ELSIF VAR_Machine.iq_stCmd.i_xAxisPhaseShift THEN
			IF 	VAR_Machine.iq_stParameter.i_uiAxisSelected >= CST_InletSubModuleHmiStart AND
				VAR_Machine.iq_stParameter.i_uiAxisSelected <= CST_InletSubModuleHmiStart + CST_LastInletModuleAxis	THEN

				VAR_Machine.stInletModule.iq_stParameters.i_uiAxisSelected		:= VAR_Machine.iq_stParameter.i_uiAxisSelected - CST_InletSubModuleHmiStart;
				VAR_Machine.stInletModule.iq_stParameters.i_rPhaseShiftDistance	:=	LREAL_TO_REAL(FC_TeensOfmmToDegrees(VAR_Machine.iq_stParameter.i_iAxisPhaseShiftDistance, CFG_MC.Mechanical.MachineStep, TRUE, FALSE));

				uiInletMultiStep	:=	600;
			END_IF
		END_IF

	545:
		IF VAR_Machine.stInletModule.iq_stStatus.q_xModuleStopped THEN
			uiInletMultiStep	:=	550;
		END_IF

	550:
		IF MC_InputOutput.Network.Inlet.Commands.StartInletModule THEN
			VAR_Machine.stInletModule.iq_stCmd.i_xStart	:= TRUE;
			uiInletMultiStep	:=	540;
		ELSIF VAR_Machine.stMasterModule.iq_stStatus.q_xSynchroWithOffset OR VAR_Machine.stInletModule.iq_stStatus.q_xSynchroWithOffset	THEN
			uiInletMultiStep	:= 800;
		END_IF

	600:
		VAR_Machine.stInletModule.iq_stCmd.i_xPhaseShift := TRUE;
		uiInletMultiStep := 610;

	610:
		IF VAR_Machine.stInletModule.iq_stStatus.q_xPhaseShiftDone AND NOT VAR_Machine.iq_stCmd.i_xAxisPhaseShift THEN
			VAR_Machine.stInletModule.iq_stCmd.i_xPhaseShift	:= FALSE;
			uiInletMultiStep	:= 540;
		END_IF

	800:
		VAR_Machine.stInletModule.iq_stCmd.i_xPhaseCompensation	:= VAR_Machine.stInletModule.iq_stStatus.q_xSynchroWithOffset;
		uiInletMultiStep	:= 810;

	810:
		IF NOT VAR_Machine.stInletModule.iq_stStatus.q_xSynchroWithOffset	THEN
			VAR_Machine.stInletModule.iq_stCmd.i_xPhaseCompensation	:= FALSE;
			uiInletMultiStep	:= 550;
		END_IF

	1000:
		IF VAR_Machine.stInletModule.iq_stStatus.q_xModuleStopped THEN
			VAR_Machine.stInletModule.iq_stCmd.i_xJogMultiMode	:= FALSE;
			VAR_Machine.stInletModule.iq_stCmd.i_xAutoMultiMode	:= FALSE;
			uiInletMultiStep	:=	0;
		END_IF

		VAR_Machine.stInletModule.iq_stCmd.i_xPhaseShift				:= FALSE;
		VAR_Machine.stInletModule.iq_stCmd.i_xStart						:= FALSE;
		VAR_Machine.stInletModule.iq_stCmd.i_xAutoMultiMode				:= FALSE;
		VAR_Machine.stInletModule.iq_stCmd.i_xJogPB						:= FALSE;
		VAR_Machine.stInletModule.iq_stCmd.i_xJogMultiMode				:= FALSE;
		VAR_Machine.stInletModule.iq_stCmd.i_xMasterRephasingRequest	:= FALSE;
		VAR_Machine.stInletModule.iq_stCmd.i_xPhaseCompensation			:= FALSE;
		VAR_Machine.stInletModule.iq_stCmd.i_xSlowMotionForward			:= FALSE;
		VAR_Machine.stInletModule.iq_stCmd.i_xSlowMotionBackward		:= FALSE;
END_CASE

xReactionOnOutletModule	:= xReactOutletEmergencyStop	OR xReactOutletQuickStop		OR xReactOutletStop			OR NOT xInputMulti OR
							(uiOutletMultiStep >= 100	AND uiOutletMultiStep < 200 	AND NOT MC_InputOutput.Network.Outlet.Commands.JogOutletModule) OR
							(uiOutletMultiStep >= 200	AND uiOutletMultiStep < 500 	AND NOT xSlowMotionCommandOutlet)	OR
							(uiOutletMultiStep >= 500	AND uiOutletMultiStep < 900 	AND NOT MC_InputOutput.Network.Outlet.Commands.AutoOutletModule);

IF xReactionOnOutletModule THEN
	IF uiOutletMultiStep <> 1000 AND uiOutletMultiStep <> 0 THEN
		uiOutletMultiStep	:=	1000;
	END_IF
END_IF

CASE uiOutletMultiStep OF
	0:(* Modality selecetion *)
		IF NOT xReactionOnOutletModule THEN
			IF MC_InputOutput.Network.Outlet.Commands.JogOutletModule AND NOT xSlowMotionCommandOutlet THEN
				uiOutletMultiStep	:=	100;
			ELSIF NOT MC_InputOutput.Network.Outlet.Commands.JogOutletModule AND xSlowMotionCommandOutlet THEN
				uiOutletMultiStep	:=	200;
			ELSIF MC_InputOutput.Network.Outlet.Commands.AutoOutletModule THEN
				uiOutletMultiStep	:=	500;
			END_IF
		END_IF

	100:(* Jog Multy *)
		VAR_Machine.stOutletModule.iq_stCmd.i_xJogMultiMode := TRUE;
		uiOutletMultiStep	:=	110;

	110:(* Wait for jog active on Outlet module and axes without offset *)
		IF VAR_Machine.stOutletModule.iq_stStatus.q_xJogMultiActive THEN
			IF NOT VAR_Machine.stOutletModule.iq_stStatus.q_xSynchroWithOffset THEN
				VAR_Machine.stOutletModule.iq_stCmd.i_xMasterRephasingRequest		:= TRUE;
				VAR_Machine.stOutletModule.iq_stParameters.i_lrRephasingPosition	:= FC_RephasingPositionOutlet(iq_astSubModuleAxis := VAR_Machine.stOutletModule.iq_astSubModuleAxis);
				VAR_Machine.iq_stCmd.i_xStart										:= TRUE;
				uiOutletMultiStep	:=	120;
			END_IF
		END_IF

	120:(* Rephasing of master position *)
		IF  VAR_Machine.stOutletModule.iq_stStatus.q_xMasterRephased THEN
			VAR_Machine.stOutletModule.iq_stCmd.i_xMasterRephasingRequest	:= FALSE;
			uiOutletMultiStep	:=	130;
		END_IF

	130:(* Jog Push button *)
		VAR_Machine.stOutletModule.iq_stCmd.i_xJogPB := MC_InputOutput.Network.Outlet.Commands.JogPushButtonOutletModule;

		IF VAR_Machine.stOutletModule.iq_stCmd.i_xJogPB THEN
			uiOutletMultiStep	:=	140;
		END_IF

	140:
		VAR_Machine.stOutletModule.iq_stCmd.i_xJogPB :=	MC_InputOutput.Network.Outlet.Commands.JogPushButtonOutletModule;
		IF NOT VAR_Machine.stOutletModule.iq_stCmd.i_xJogPB THEN
			VAR_Machine.stOutletModule.iq_stCmd.i_xJogMultiMode	:= FALSE;
			uiOutletMultiStep	:=	160;
		END_IF

	160:
		IF VAR_Machine.stOutletModule.iq_stStatus.q_xModuleStopped AND NOT VAR_Machine.stOutletModule.iq_stStatus.q_xJogMultiActive	THEN
			uiOutletMultiStep	:=	100;
		END_IF

	200:
		VAR_Machine.stOutletModule.iq_stCmd.i_xSlowMotionForward	:= xSlowMotionCommandOutletForward;
		VAR_Machine.stOutletModule.iq_stCmd.i_xSlowMotionBackward	:= xSlowMotionCommandOutletBackward;
		uiOutletMultiStep	:=	230;

	230:
		IF VAR_Machine.stOutletModule.iq_stStatus.q_xSlowMotionActive THEN
			uiOutletMultiStep	:=	250;
		END_IF

	250:
		VAR_Machine.stOutletModule.iq_stCmd.i_xSlowMotionForward	:= xSlowMotionCommandOutletForward;
		VAR_Machine.stOutletModule.iq_stCmd.i_xSlowMotionBackward	:= xSlowMotionCommandOutletBackward;
		VAR_Machine.stOutletModule.iq_stCmd.i_xJogPB				:= MC_InputOutput.Network.Outlet.Commands.JogPushButtonOutletModule;

	500:
		VAR_Machine.stOutletModule.iq_stCmd.i_xAutoMultiMode := TRUE;
		uiOutletMultiStep	:=	510;

	510:(* The phase compensation process has to be ended bofore going on next steps *)
		IF VAR_Machine.stOutletModule.iq_stStatus.q_xAutoMultiActive THEN
			IF NOT VAR_Machine.stOutletModule.iq_stStatus.q_xSynchroWithOffset THEN
				VAR_Machine.stOutletModule.iq_stParameters.i_lrRephasingPosition	:= FC_RephasingPositionOutlet(iq_astSubModuleAxis := VAR_Machine.stOutletModule.iq_astSubModuleAxis);
				uiOutletMultiStep	:=	520;
			END_IF
		END_IF

	520:(* Rephasing position of the master *)
		VAR_Machine.stOutletModule.iq_stCmd.i_xMasterRephasingRequest	:= TRUE;
		IF  VAR_Machine.stOutletModule.iq_stStatus.q_xMasterRephased THEN
			VAR_Machine.stOutletModule.iq_stCmd.i_xMasterRephasingRequest := FALSE;
			uiOutletMultiStep	:=	530;
		END_IF

	530:(* Wait the start command from the plc *)
		IF MC_InputOutput.Network.Outlet.Commands.StartOutletModule THEN
			VAR_Machine.stOutletModule.iq_stCmd.i_xStart := TRUE;
			uiOutletMultiStep := 540;
		END_IF

	540:
		IF NOT MC_InputOutput.Network.Outlet.Commands.StartOutletModule THEN
			VAR_Machine.stOutletModule.iq_stCmd.i_xStart := FALSE;
			uiOutletMultiStep := 545;
		ELSIF VAR_Machine.iq_stCmd.i_xAxisPhaseShift THEN
			IF VAR_Machine.iq_stParameter.i_uiAxisSelected >= CST_OutletSubModuleHmiStart AND
				VAR_Machine.iq_stParameter.i_uiAxisSelected <= CST_OutletSubModuleHmiStart + CST_LastOutletModuleAxis THEN

				VAR_Machine.stOutletModule.iq_stParameters.i_uiAxisSelected			:= VAR_Machine.iq_stParameter.i_uiAxisSelected - CST_OutletSubModuleHmiStart;
				VAR_Machine.stOutletModule.iq_stParameters.i_rPhaseShiftDistance	:=	LREAL_TO_REAL(FC_TeensOfmmToDegrees(VAR_Machine.iq_stParameter.i_iAxisPhaseShiftDistance, CFG_MC.Mechanical.MachineStep, TRUE, FALSE));
				uiOutletMultiStep	:=	600;
			END_IF
		END_IF

	545:
		IF VAR_Machine.stOutletModule.iq_stStatus.q_xModuleStopped THEN
			uiOutletMultiStep	:=	550;
		END_IF

	550:
		IF MC_InputOutput.Network.Outlet.Commands.StartOutletModule THEN
			VAR_Machine.stOutletModule.iq_stCmd.i_xStart := TRUE;
			uiOutletMultiStep := 540;
		ELSIF VAR_Machine.stMasterModule.iq_stStatus.q_xSynchroWithOffset OR
			VAR_Machine.stOutletModule.iq_stStatus.q_xSynchroWithOffset	THEN
			uiOutletMultiStep	:= 800;
		END_IF

	600:
		VAR_Machine.stOutletModule.iq_stCmd.i_xPhaseShift := TRUE;
		uiOutletMultiStep	:= 610;

	610:
		IF VAR_Machine.stOutletModule.iq_stStatus.q_xPhaseShiftDone AND NOT VAR_Machine.iq_stCmd.i_xAxisPhaseShift THEN
			VAR_Machine.stOutletModule.iq_stCmd.i_xPhaseShift := FALSE;
			uiOutletMultiStep	:= 540;
		END_IF

	800:
		VAR_Machine.stOutletModule.iq_stCmd.i_xPhaseCompensation	:= VAR_Machine.stOutletModule.iq_stStatus.q_xSynchroWithOffset;
		uiOutletMultiStep	:= 810;

	810:
		IF NOT VAR_Machine.stOutletModule.iq_stStatus.q_xSynchroWithOffset THEN
			VAR_Machine.stOutletModule.iq_stCmd.i_xPhaseCompensation := FALSE;
			uiOutletMultiStep	:= 550;
		END_IF

	1000:
		IF VAR_Machine.stOutletModule.iq_stStatus.q_xModuleStopped THEN
			VAR_Machine.stOutletModule.iq_stCmd.i_xJogMultiMode		:= FALSE;
			VAR_Machine.stOutletModule.iq_stCmd.i_xAutoMultiMode	:= FALSE;
			uiOutletMultiStep	:=	0;
		END_IF

		VAR_Machine.stOutletModule.iq_stCmd.i_xPhaseShift				:= FALSE;
		VAR_Machine.stOutletModule.iq_stCmd.i_xStart					:= FALSE;
		VAR_Machine.stOutletModule.iq_stCmd.i_xAutoMultiMode			:= FALSE;
		VAR_Machine.stOutletModule.iq_stCmd.i_xJogPB					:= FALSE;
		VAR_Machine.stOutletModule.iq_stCmd.i_xJogMultiMode				:= FALSE;
		VAR_Machine.stOutletModule.iq_stCmd.i_xMasterRephasingRequest	:= FALSE;
		VAR_Machine.stOutletModule.iq_stCmd.i_xPhaseCompensation		:= FALSE;
		VAR_Machine.stOutletModule.iq_stCmd.i_xSlowMotionForward		:= FALSE;
		VAR_Machine.stOutletModule.iq_stCmd.i_xSlowMotionBackward		:= FALSE;
END_CASE
END_STEP
ENTRY_ACTION
uiFillerMultiStep	:=	0;
uiInletMultiStep	:=	0;
uiOutletMultiStep	:=	0;
END_ACTION
EXIT_ACTION
VAR_Machine.stFillerModule.iq_stCmd.i_xMasterRephasingRequest	:=	FALSE;
VAR_Machine.stOutletModule.iq_stCmd.i_xMasterRephasingRequest	:=	FALSE;
VAR_Machine.stInletModule.iq_stCmd.i_xMasterRephasingRequest	:=	FALSE;
END_ACTION
TRANSITION FROM Multi TO MultiExit:=
NOT xMultiMode
END_TRANSITION
STEP MultiExit:
IF NOT VAR_Machine.stFillerModule.iq_stStatus.q_xAutoMultiActive		AND
	NOT VAR_Machine.stFillerModule.iq_stStatus.q_xJogMultiActive		AND

	((NOT VAR_Machine.stInletModule.iq_stStatus.q_xAutoMultiActive 		AND
	NOT VAR_Machine.stInletModule.iq_stStatus.q_xJogMultiActive)		OR NOT
	VAR_Machine.stInletModule.iq_stStatus.q_xModuleReal)				AND

	((NOT VAR_Machine.stOutletModule.iq_stStatus.q_xAutoMultiActive		AND
	NOT VAR_Machine.stOutletModule.iq_stStatus.q_xJogMultiActive)		OR NOT
	VAR_Machine.stOutletModule.iq_stStatus.q_xModuleReal)				THEN

	xExitStep	:= TRUE;
END_IF
END_STEP
ENTRY_ACTION
VAR_Machine.stFillerModule.iq_stCmd.i_xPhaseShift				:= FALSE;
VAR_Machine.stInletModule.iq_stCmd.i_xPhaseShift				:= FALSE;
VAR_Machine.stOutletModule.iq_stCmd.i_xPhaseShift				:= FALSE;

VAR_Machine.stFillerModule.iq_stCmd.i_xStart					:= FALSE;
VAR_Machine.stInletModule.iq_stCmd.i_xStart						:= FALSE;
VAR_Machine.stOutletModule.iq_stCmd.i_xStart					:= FALSE;

VAR_Machine.stFillerModule.iq_stCmd.i_xAutoMultiMode			:= FALSE;
VAR_Machine.stInletModule.iq_stCmd.i_xAutoMultiMode				:= FALSE;
VAR_Machine.stOutletModule.iq_stCmd.i_xAutoMultiMode			:= FALSE;

VAR_Machine.stFillerModule.iq_stCmd.i_xJogPB					:= FALSE;
VAR_Machine.stInletModule.iq_stCmd.i_xJogPB						:= FALSE;
VAR_Machine.stOutletModule.iq_stCmd.i_xJogPB					:= FALSE;

VAR_Machine.stFillerModule.iq_stCmd.i_xJogMultiMode				:= FALSE;
VAR_Machine.stInletModule.iq_stCmd.i_xJogMultiMode				:= FALSE;
VAR_Machine.stOutletModule.iq_stCmd.i_xJogMultiMode				:= FALSE;

VAR_Machine.stFillerModule.iq_stCmd.i_xMasterRephasingRequest	:= FALSE;
VAR_Machine.stInletModule.iq_stCmd.i_xMasterRephasingRequest	:= FALSE;
VAR_Machine.stOutletModule.iq_stCmd.i_xMasterRephasingRequest	:= FALSE;

VAR_Machine.stFillerModule.iq_stCmd.i_xPhaseCompensation		:= FALSE;
VAR_Machine.stInletModule.iq_stCmd.i_xPhaseCompensation			:= FALSE;
VAR_Machine.stOutletModule.iq_stCmd.i_xPhaseCompensation		:= FALSE;

VAR_Machine.stInletModule.iq_stCmd.i_xSlowMotionForward			:= FALSE;
VAR_Machine.stInletModule.iq_stCmd.i_xSlowMotionBackward		:= FALSE;

VAR_Machine.stOutletModule.iq_stCmd.i_xSlowMotionForward		:= FALSE;
VAR_Machine.stOutletModule.iq_stCmd.i_xSlowMotionBackward		:= FALSE;

xEncEmulationEnable	:= FALSE;
END_ACTION
TRANSITION FROM MultiExit TO ModeSelection:=
xExitStep
END_TRANSITION
(* @SFCISJUMP := 'ModeSelection' *)
TRANSITION FROM ModeSelection TO Jog:=
xJogMode
END_TRANSITION
STEP Jog:
IF xReactionActive OR NOT xInputJog THEN
	xJogMode := FALSE;
END_IF

xJogActive	:= TRUE;

CASE uiJogStep OF
	0:
		VAR_Machine.stFillerModule.iq_stCmd.i_xAutoMode	:= TRUE;
		VAR_Machine.stOutletModule.iq_stCmd.i_xAutoMode	:= VAR_Machine.stOutletModule.iq_stStatus.q_xModuleReal;
		VAR_Machine.stInletModule.iq_stCmd.i_xAutoMode	:= VAR_Machine.stInletModule.iq_stStatus.q_xModuleReal;
		uiJogStep	:=	40;

	40:
		IF VAR_Machine.stFillerModule.iq_stStatus.q_xAutoActive		AND
			(VAR_Machine.stOutletModule.iq_stStatus.q_xAutoActive	OR NOT
			VAR_Machine.stOutletModule.iq_stStatus.q_xModuleReal)	AND
			(VAR_Machine.stInletModule.iq_stStatus.q_xAutoActive	OR NOT
			VAR_Machine.stInletModule.iq_stStatus.q_xModuleReal)	THEN

			IF NOT VAR_Machine.stFillerModule.iq_stStatus.q_xSynchroWithOffset		AND
				NOT VAR_Machine.stOutletModule.iq_stStatus.q_xSynchroWithOffset		AND
				NOT VAR_Machine.stInletModule.iq_stStatus.q_xSynchroWithOffset		THEN

				VAR_Machine.stMasterModule.iq_stParameters.i_lrRephasingPosition :=
								FC_RephasingMachine(iq_astInletSubModuleAxis	:= VAR_Machine.stInletModule.iq_astSubModuleAxis,
													iq_astFillerSubModuleAxis	:= VAR_Machine.stFillerModule.iq_astSubModuleAxis,
													iq_astOutletSubModuleAxis	:= VAR_Machine.stOutletModule.iq_astSubModuleAxis);

				VAR_Machine.stFillerModule.iq_stParameters.i_lrRephasingPosition
					:=	VAR_Machine.stMasterModule.iq_stParameters.i_lrRephasingPosition;

				VAR_Machine.stOutletModule.iq_stParameters.i_lrRephasingPosition
					:=	VAR_Machine.stMasterModule.iq_stParameters.i_lrRephasingPosition;

				VAR_Machine.stInletModule.iq_stParameters.i_lrRephasingPosition
					:=	VAR_Machine.stMasterModule.iq_stParameters.i_lrRephasingPosition;

				uiJogStep	:=	100;
			END_IF
		END_IF

	100:
		VAR_Machine.stMasterModule.iq_stCmd.i_xMasterRephasingRequest	:= 	TRUE;
		VAR_Machine.stMasterModule.iq_stCmd.i_xJogMode					:=	TRUE;

		IF VAR_Machine.stMasterModule.iq_stStatus.q_xJogActive AND VAR_Machine.stMasterModule.iq_stStatus.q_xMasterRephased THEN
			VAR_Machine.stMasterModule.iq_stCmd.i_xMasterRephasingRequest	:= FALSE;
			uiJogStep	:=	110;
		END_IF

	110:
		IF VAR_Machine.iq_stCmd.i_xJogPushButton THEN
			VAR_Machine.stFillerModule.iq_stCmd.i_xStart	:=	TRUE;
			VAR_Machine.stOutletModule.iq_stCmd.i_xStart	:=	VAR_Machine.stOutletModule.iq_stStatus.q_xModuleReal;
			VAR_Machine.stInletModule.iq_stCmd.i_xStart		:=	VAR_Machine.stInletModule.iq_stStatus.q_xModuleReal;
			uiJogStep	:=	120;
		END_IF

	120:
		IF VAR_Machine.stFillerModule.iq_stStatus.q_xRealAxesSynchronized		AND
			VAR_Machine.stFillerModule.iq_stStatus.q_xAutoActive				AND

			((VAR_Machine.stInletModule.iq_stStatus.q_xRealAxesSynchronized		AND
			VAR_Machine.stInletModule.iq_stStatus.q_xAutoActive)				OR NOT
			VAR_Machine.stInletModule.iq_stStatus.q_xModuleReal)				AND

			((VAR_Machine.stOutletModule.iq_stStatus.q_xRealAxesSynchronized	AND
			VAR_Machine.stOutletModule.iq_stStatus.q_xAutoActive)				OR NOT
			VAR_Machine.stOutletModule.iq_stStatus.q_xModuleReal)				THEN

			VAR_Machine.stMasterModule.iq_stCmd.i_xJogPB :=	VAR_Machine.iq_stCmd.i_xJogPushButton;
			xEncEmulationEnable	:= TRUE;
			uiJogStep	:=	130;
		END_IF

	130:
		VAR_Machine.stMasterModule.iq_stCmd.i_xJogPB :=	VAR_Machine.iq_stCmd.i_xJogPushButton;
		IF NOT VAR_Machine.iq_stCmd.i_xJogPushButton THEN
			VAR_Machine.stMasterModule.iq_stCmd.i_xJogPB	:= FALSE;
			uiJogStep	:= 135;
		ELSIF VAR_Machine.iq_stCmd.i_xAxisPhaseShift THEN
			IF VAR_Machine.iq_stParameter.i_uiAxisSelected >= CST_FillerSubModuleHmiStart AND
				VAR_Machine.iq_stParameter.i_uiAxisSelected <= CST_FillerSubModuleHmiStart + CST_LastFillerModuleAxis	THEN

				VAR_Machine.stFillerModule.iq_stParameters.i_uiAxisSelected
					:=	VAR_Machine.iq_stParameter.i_uiAxisSelected - CST_FillerSubModuleHmiStart;

				VAR_Machine.stFillerModule.iq_stParameters.i_rPhaseShiftDistance
					:=	LREAL_TO_REAL(FC_TeensOfmmToDegrees(VAR_Machine.iq_stParameter.i_iAxisPhaseShiftDistance, CFG_MC.Mechanical.MachineStep, TRUE, FALSE));

				uiJogStep	:=	200;
			ELSIF VAR_Machine.iq_stParameter.i_uiAxisSelected >= CST_OutletSubModuleHmiStart AND
				VAR_Machine.iq_stParameter.i_uiAxisSelected <= CST_OutletSubModuleHmiStart + CST_LastOutletModuleAxis THEN

				VAR_Machine.stOutletModule.iq_stParameters.i_uiAxisSelected
					:=	VAR_Machine.iq_stParameter.i_uiAxisSelected - CST_OutletSubModuleHmiStart;

				VAR_Machine.stOutletModule.iq_stParameters.i_rPhaseShiftDistance
					:=	LREAL_TO_REAL(FC_TeensOfmmToDegrees(VAR_Machine.iq_stParameter.i_iAxisPhaseShiftDistance, CFG_MC.Mechanical.MachineStep, TRUE, FALSE));

				uiJogStep	:=	300;
			ELSIF VAR_Machine.iq_stParameter.i_uiAxisSelected >= CST_InletSubModuleHmiStart AND
				VAR_Machine.iq_stParameter.i_uiAxisSelected <= CST_InletSubModuleHmiStart + CST_LastInletModuleAxis THEN

				VAR_Machine.stInletModule.iq_stParameters.i_uiAxisSelected
					:=	VAR_Machine.iq_stParameter.i_uiAxisSelected - CST_InletSubModuleHmiStart;

				VAR_Machine.stInletModule.iq_stParameters.i_rPhaseShiftDistance
					:=	LREAL_TO_REAL(FC_TeensOfmmToDegrees(VAR_Machine.iq_stParameter.i_iAxisPhaseShiftDistance, CFG_MC.Mechanical.MachineStep, TRUE, FALSE));

				uiJogStep	:=	400;
			END_IF
		END_IF

	135:
		IF VAR_Machine.stMasterModule.iq_stStatus.q_xModuleStopped THEN
			xEncEmulationEnable	:= FALSE;
			uiJogStep	:=	140;
		END_IF

	140:
		IF VAR_Machine.iq_stCmd.i_xJogPushButton THEN
			uiJogStep	:=	120;
		ELSIF VAR_Machine.stMasterModule.iq_stStatus.q_xSynchroWithOffset	OR
			VAR_Machine.stFillerModule.iq_stStatus.q_xSynchroWithOffset		OR
			(VAR_Machine.stOutletModule.iq_stStatus.q_xSynchroWithOffset	AND
			VAR_Machine.stOutletModule.iq_stStatus.q_xModuleReal)			OR
			(VAR_Machine.stInletModule.iq_stStatus.q_xSynchroWithOffset		AND
			VAR_Machine.stInletModule.iq_stStatus.q_xModuleReal)			THEN

			uiJogStep	:= 800;

		END_IF

	200:
		VAR_Machine.stFillerModule.iq_stCmd.i_xPhaseShift	:= TRUE;
		uiJogStep	:= 210;

	210:
		IF VAR_Machine.stFillerModule.iq_stStatus.q_xPhaseShiftDone AND NOT VAR_Machine.iq_stCmd.i_xAxisPhaseShift THEN
			VAR_Machine.stFillerModule.iq_stCmd.i_xPhaseShift	:= FALSE;
			uiJogStep	:= 130;
		END_IF

	300:
		VAR_Machine.stOutletModule.iq_stCmd.i_xPhaseShift	:= TRUE;
		uiJogStep	:= 310;

	310:
		IF VAR_Machine.stOutletModule.iq_stStatus.q_xPhaseShiftDone AND NOT VAR_Machine.iq_stCmd.i_xAxisPhaseShift THEN
			VAR_Machine.stOutletModule.iq_stCmd.i_xPhaseShift	:= FALSE;
			uiJogStep	:= 130;
		END_IF

	400:
		VAR_Machine.stInletModule.iq_stCmd.i_xPhaseShift	:= TRUE;
		uiJogStep	:= 410;

	410:
		IF VAR_Machine.stInletModule.iq_stStatus.q_xPhaseShiftDone AND NOT VAR_Machine.iq_stCmd.i_xAxisPhaseShift THEN
			VAR_Machine.stInletModule.iq_stCmd.i_xPhaseShift	:= FALSE;
			uiJogStep	:= 130;
		END_IF

	800:
		VAR_Machine.stMasterModule.iq_stCmd.i_xPhaseCompensation	:= VAR_Machine.stMasterModule.iq_stStatus.q_xSynchroWithOffset;
		VAR_Machine.stFillerModule.iq_stCmd.i_xPhaseCompensation	:= VAR_Machine.stFillerModule.iq_stStatus.q_xSynchroWithOffset;
		VAR_Machine.stOutletModule.iq_stCmd.i_xPhaseCompensation	:= VAR_Machine.stOutletModule.iq_stStatus.q_xSynchroWithOffset;
		VAR_Machine.stInletModule.iq_stCmd.i_xPhaseCompensation		:= VAR_Machine.stInletModule.iq_stStatus.q_xSynchroWithOffset;
		uiJogStep	:= 810;

	810:
		IF NOT VAR_Machine.stMasterModule.iq_stStatus.q_xSynchroWithOffset		AND
			NOT VAR_Machine.stFillerModule.iq_stStatus.q_xSynchroWithOffset		AND
			(NOT VAR_Machine.stOutletModule.iq_stStatus.q_xSynchroWithOffset	OR
			NOT VAR_Machine.stOutletModule.iq_stStatus.q_xModuleReal)			AND
			(NOT VAR_Machine.stInletModule.iq_stStatus.q_xSynchroWithOffset		OR
			NOT VAR_Machine.stInletModule.iq_stStatus.q_xModuleReal)			THEN

			VAR_Machine.stMasterModule.iq_stCmd.i_xPhaseCompensation	:= FALSE;
			VAR_Machine.stFillerModule.iq_stCmd.i_xPhaseCompensation	:= FALSE;
			VAR_Machine.stOutletModule.iq_stCmd.i_xPhaseCompensation	:= FALSE;
			VAR_Machine.stInletModule.iq_stCmd.i_xPhaseCompensation		:= FALSE;
			uiJogStep	:= 140;
		END_IF
END_CASE
END_STEP
ENTRY_ACTION
uiJogStep	:=	0;
END_ACTION
TRANSITION FROM Jog TO JogExit:=
NOT xJogMode
END_TRANSITION
STEP JogExit:
IF NOT VAR_Machine.stMasterModule.iq_stStatus.q_xJogActive		AND
	NOT VAR_Machine.stFillerModule.iq_stStatus.q_xAutoActive	AND
	(NOT VAR_Machine.stOutletModule.iq_stStatus.q_xAutoActive	OR NOT
	VAR_Machine.stOutletModule.iq_stStatus.q_xModuleReal)		AND
	(NOT VAR_Machine.stInletModule.iq_stStatus.q_xAutoActive	OR NOT
	VAR_Machine.stInletModule.iq_stStatus.q_xModuleReal)		THEN

	xExitStep	:= TRUE;
END_IF
END_STEP
ENTRY_ACTION
VAR_Machine.stFillerModule.iq_stCmd.i_xPhaseShift				:= FALSE;
VAR_Machine.stOutletModule.iq_stCmd.i_xPhaseShift				:= FALSE;
VAR_Machine.stInletModule.iq_stCmd.i_xPhaseShift				:= FALSE;

VAR_Machine.stMasterModule.iq_stCmd.i_xStart					:= FALSE;
VAR_Machine.stFillerModule.iq_stCmd.i_xStart					:= FALSE;
VAR_Machine.stOutletModule.iq_stCmd.i_xStart					:= FALSE;
VAR_Machine.stInletModule.iq_stCmd.i_xStart						:= FALSE;

VAR_Machine.stMasterModule.iq_stCmd.i_xJogMode					:= FALSE;
VAR_Machine.stFillerModule.iq_stCmd.i_xAutoMode					:= FALSE;
VAR_Machine.stOutletModule.iq_stCmd.i_xAutoMode					:= FALSE;
VAR_Machine.stInletModule.iq_stCmd.i_xAutoMode					:= FALSE;
VAR_Machine.stMasterModule.iq_stCmd.i_xMasterRephasingRequest	:= FALSE;

VAR_Machine.stMasterModule.iq_stCmd.i_xJogPB					:= FALSE;

xEncEmulationEnable	:= FALSE;
END_ACTION
TRANSITION FROM JogExit TO ModeSelection:=
xExitStep
END_TRANSITION
(* @SFCISJUMP := 'ModeSelection' *)
TRANSITION FROM ModeSelection TO BrakeRelease:=
xBrakeReleaseMode
END_TRANSITION
STEP BrakeRelease:
IF NOT tofReactionActive.Q THEN
	xBrakeReleaseMode	:= FALSE;
END_IF

xBrakeReleaseActive	:= TRUE;

CASE uiBrakeReleaseStep OF
	0:
		IF xInputBrakeRelease THEN
			uiOldAxisSelected	:= VAR_Machine.iq_stParameter.i_uiAxisSelected;
			IF 	VAR_Machine.iq_stParameter.i_uiAxisSelected >= CST_FillerSubModuleHmiStart AND
				VAR_Machine.iq_stParameter.i_uiAxisSelected <= CST_FillerSubModuleHmiStart + CST_LastFillerModuleAxis	THEN

				VAR_Machine.stFillerModule.iq_stParameters.i_uiAxisSelected	:= VAR_Machine.iq_stParameter.i_uiAxisSelected - CST_FillerSubModuleHmiStart;
				uiBrakeReleaseStep	:= 100;
			ELSIF 	VAR_Machine.iq_stParameter.i_uiAxisSelected >= CST_OutletSubModuleHmiStart AND
				VAR_Machine.iq_stParameter.i_uiAxisSelected <= CST_OutletSubModuleHmiStart + CST_LastOutletModuleAxis THEN

				VAR_Machine.stOutletModule.iq_stParameters.i_uiAxisSelected	:= VAR_Machine.iq_stParameter.i_uiAxisSelected - CST_OutletSubModuleHmiStart;
				uiBrakeReleaseStep	:= 300;

			ELSIF 	VAR_Machine.iq_stParameter.i_uiAxisSelected >= CST_InletSubModuleHmiStart AND
				VAR_Machine.iq_stParameter.i_uiAxisSelected <= CST_InletSubModuleHmiStart + CST_LastInletModuleAxis THEN

				VAR_Machine.stInletModule.iq_stParameters.i_uiAxisSelected	:= VAR_Machine.iq_stParameter.i_uiAxisSelected - CST_InletSubModuleHmiStart;
				uiBrakeReleaseStep	:= 600;
			END_IF
		ELSE
			xBrakeReleaseMode	:= FALSE;
		END_IF

	100:(* Brake Release On Filler Module *)
		VAR_Machine.stFillerModule.iq_stCmd.i_xBrakeRelease := TRUE;
		IF VAR_Machine.stFillerModule.iq_stStatus.q_xBrakeReleaseDone THEN
			uiBrakeReleaseStep	:= 150;
		END_IF

	150:
		IF uiOldAxisSelected <> VAR_Machine.iq_stParameter.i_uiAxisSelected THEN
			VAR_Machine.stFillerModule.iq_stCmd.i_xBrakeRelease := FALSE;
			uiBrakeReleaseStep		:= 160;
		ELSIF NOT xInputBrakeRelease THEN
			uiBrakeReleaseStep		:= 190;
		END_IF

	160:
		IF NOT VAR_Machine.stFillerModule.iq_stStatus.q_xBrakeReleaseActive AND NOT VAR_Machine.stFillerModule.iq_stStatus.q_xBrakeReleaseDone THEN
			uiBrakeReleaseStep	:= 0;
		END_IF

	190:
		IF uiOldAxisSelected <> VAR_Machine.iq_stParameter.i_uiAxisSelected THEN
			VAR_Machine.stFillerModule.iq_stCmd.i_xBrakeRelease := FALSE;
			uiBrakeReleaseStep		:= 160;
		ELSIF xInputBrakeRelease THEN
			VAR_Machine.stFillerModule.iq_stCmd.i_xBrakeRelease := FALSE;
			uiBrakeReleaseStep		:= 200;
		END_IF

	200:
		IF NOT VAR_Machine.stFillerModule.iq_stStatus.q_xBrakeReleaseActive AND NOT VAR_Machine.stFillerModule.iq_stStatus.q_xBrakeReleaseDone AND NOT xInputBrakeRelease THEN
			xBrakeReleaseMode	:= FALSE;
		END_IF

	300:(* Brake Release On Outlet Module *)
		VAR_Machine.stOutletModule.iq_stCmd.i_xBrakeRelease := TRUE;
		IF VAR_Machine.stOutletModule.iq_stStatus.q_xBrakeReleaseDone THEN
			uiBrakeReleaseStep	:= 350;
		END_IF

	350:
		IF uiOldAxisSelected <> VAR_Machine.iq_stParameter.i_uiAxisSelected THEN
			VAR_Machine.stOutletModule.iq_stCmd.i_xBrakeRelease := FALSE;
			uiBrakeReleaseStep		:= 360;
		ELSIF NOT xInputBrakeRelease THEN
			VAR_Machine.stOutletModule.iq_stCmd.i_xBrakeRelease := FALSE;
			uiBrakeReleaseStep		:= 390;
		END_IF

	360:
		IF NOT VAR_Machine.stOutletModule.iq_stStatus.q_xBrakeReleaseActive AND NOT VAR_Machine.stOutletModule.iq_stStatus.q_xBrakeReleaseDone THEN
			uiBrakeReleaseStep	:= 0;
		END_IF

	390:
		IF uiOldAxisSelected <> VAR_Machine.iq_stParameter.i_uiAxisSelected THEN
			VAR_Machine.stOutletModule.iq_stCmd.i_xBrakeRelease := FALSE;
			uiBrakeReleaseStep		:= 360;
		ELSIF xInputBrakeRelease THEN
			VAR_Machine.stOutletModule.iq_stCmd.i_xBrakeRelease := FALSE;
			uiBrakeReleaseStep		:= 400;
		END_IF

	400:
		IF NOT VAR_Machine.stOutletModule.iq_stStatus.q_xBrakeReleaseActive AND NOT VAR_Machine.stOutletModule.iq_stStatus.q_xBrakeReleaseDone  AND NOT xInputBrakeRelease THEN
			xBrakeReleaseMode	:= FALSE;
		END_IF

	600:(* Brake Release On Inlet Module *)
		VAR_Machine.stInletModule.iq_stCmd.i_xBrakeRelease := TRUE;
		IF 	VAR_Machine.stInletModule.iq_stStatus.q_xBrakeReleaseDone THEN
			uiBrakeReleaseStep	:= 650;
		END_IF

	650:
		IF uiOldAxisSelected <> VAR_Machine.iq_stParameter.i_uiAxisSelected THEN
			VAR_Machine.stInletModule.iq_stCmd.i_xBrakeRelease := FALSE;
			uiBrakeReleaseStep		:= 660;
		ELSIF NOT xInputBrakeRelease THEN
			VAR_Machine.stInletModule.iq_stCmd.i_xBrakeRelease := FALSE;
			uiBrakeReleaseStep		:= 690;
		END_IF

	660:
		IF NOT VAR_Machine.stInletModule.iq_stStatus.q_xBrakeReleaseActive AND NOT VAR_Machine.stInletModule.iq_stStatus.q_xBrakeReleaseDone THEN
			uiBrakeReleaseStep	:= 0;
		END_IF

	690:
		IF uiOldAxisSelected <> VAR_Machine.iq_stParameter.i_uiAxisSelected THEN
			VAR_Machine.stInletModule.iq_stCmd.i_xBrakeRelease := FALSE;
			uiBrakeReleaseStep		:= 660;
		ELSIF xInputBrakeRelease THEN
			VAR_Machine.stInletModule.iq_stCmd.i_xBrakeRelease := FALSE;
			uiBrakeReleaseStep		:= 700;
		END_IF

	700:
		IF NOT VAR_Machine.stInletModule.iq_stStatus.q_xBrakeReleaseActive AND NOT VAR_Machine.stInletModule.iq_stStatus.q_xBrakeReleaseDone  AND NOT xInputBrakeRelease THEN
			xBrakeReleaseMode	:= FALSE;
		END_IF
END_CASE
END_STEP
ENTRY_ACTION
uiBrakeReleaseStep	:= 0;
END_ACTION
TRANSITION FROM BrakeRelease TO BrakeExit:=
NOT xBrakeReleaseMode
END_TRANSITION
STEP BrakeExit:
xExitStep := TRUE;
END_STEP
ENTRY_ACTION
VAR_Machine.stFillerModule.iq_stCmd.i_xBrakeRelease	:= FALSE;
VAR_Machine.stInletModule.iq_stCmd.i_xBrakeRelease	:= FALSE;
VAR_Machine.stOutletModule.iq_stCmd.i_xBrakeRelease	:= FALSE;
xBrakeReleaseActive := FALSE;
END_ACTION
TRANSITION FROM BrakeExit TO ModeSelection:=
xExitStep
END_TRANSITION
(* @SFCISJUMP := 'ModeSelection' *)
TRANSITION FROM ModeSelection TO ThirdPartySetup:=
xThirdPartySetupMode
END_TRANSITION
STEP ThirdPartySetup:
IF xThirdPartySetupDone OR xReactionActive THEN
	xThirdPartySetupMode	:= FALSE;
END_IF

xThirdPartySetupActive	:= TRUE;

CASE uiThirdPartySetupStep OF
	0:
		IF	VAR_Machine.iq_stParameter.i_uiAxisSelected >= CST_FillerSubModuleHmiStart AND
			VAR_Machine.iq_stParameter.i_uiAxisSelected <= CST_FillerSubModuleHmiStart + CST_LastFillerModuleAxis	THEN

			VAR_Machine.stFillerModule.iq_stParameters.i_uiAxisSelected
				:=	VAR_Machine.iq_stParameter.i_uiAxisSelected - CST_FillerSubModuleHmiStart;

			uiThirdPartySetupStep	:=	100;
		ELSIF VAR_Machine.iq_stParameter.i_uiAxisSelected >= CST_InletSubModuleHmiStart AND
			VAR_Machine.iq_stParameter.i_uiAxisSelected <= CST_InletSubModuleHmiStart + CST_LastInletModuleAxis THEN

			VAR_Machine.stInletModule.iq_stParameters.i_uiAxisSelected
				:=	VAR_Machine.iq_stParameter.i_uiAxisSelected - CST_InletSubModuleHmiStart;

			uiThirdPartySetupStep	:=	200;
		ELSIF 	VAR_Machine.iq_stParameter.i_uiAxisSelected >= CST_OutletSubModuleHmiStart AND
			VAR_Machine.iq_stParameter.i_uiAxisSelected <= CST_OutletSubModuleHmiStart + CST_LastOutletModuleAxis THEN

			VAR_Machine.stOutletModule.iq_stParameters.i_uiAxisSelected
				:=	VAR_Machine.iq_stParameter.i_uiAxisSelected - CST_OutletSubModuleHmiStart;

			uiThirdPartySetupStep	:=	300;
		END_IF

	100:(* Third Party motor setup on Filler Module *)
		VAR_Machine.stFillerModule.iq_stCmd.i_xThirdPartySetup :=	TRUE;

		IF VAR_Machine.stFillerModule.iq_stStatus.q_xThirdPartySetupActive 	AND
			VAR_Machine.stFillerModule.iq_stStatus.q_xThirdPartySetupDone	THEN

			VAR_Machine.stFillerModule.iq_stCmd.i_xThirdPartySetup 			:=	FALSE;
			VAR_Machine.stFillerModule.iq_stParameters.i_uiAxisSelected		:=	CST_FirstFillerModuleAxis;
			uiThirdPartySetupStep	:=	150;
		END_IF

	150:
		IF NOT VAR_Machine.stFillerModule.iq_stStatus.q_xThirdPartySetupActive 	AND
			NOT VAR_Machine.stFillerModule.iq_stStatus.q_xThirdPartySetupDone	THEN
			uiThirdPartySetupStep	:=	400;
		END_IF

	200:(* Third Party motor setup on Inlet Module *)
		VAR_Machine.stInletModule.iq_stCmd.i_xThirdPartySetup :=	TRUE;

		IF VAR_Machine.stInletModule.iq_stStatus.q_xThirdPartySetupActive	AND
			VAR_Machine.stInletModule.iq_stStatus.q_xThirdPartySetupDone	THEN

			VAR_Machine.stInletModule.iq_stCmd.i_xThirdPartySetup 			:=	FALSE;
			VAR_Machine.stInletModule.iq_stParameters.i_uiAxisSelected		:=	CST_FirstInletModuleAxis;
			uiThirdPartySetupStep	:=	250;
		END_IF

	250:
		IF NOT VAR_Machine.stInletModule.iq_stStatus.q_xThirdPartySetupActive 	AND
			NOT	VAR_Machine.stInletModule.iq_stStatus.q_xThirdPartySetupDone	THEN
			uiThirdPartySetupStep	:=	400;
		END_IF

	300:(* Third Party motor setup on Outlet Module *)
		VAR_Machine.stOutletModule.iq_stCmd.i_xThirdPartySetup :=	TRUE;

		IF VAR_Machine.stOutletModule.iq_stStatus.q_xThirdPartySetupActive	AND
			VAR_Machine.stOutletModule.iq_stStatus.q_xThirdPartySetupDone	THEN

			VAR_Machine.stOutletModule.iq_stCmd.i_xThirdPartySetup 			:=	FALSE;
			VAR_Machine.stOutletModule.iq_stParameters.i_uiAxisSelected		:=	CST_FirstOutletModuleAxis;
			uiThirdPartySetupStep	:=	350;
		END_IF

	350:
		IF NOT VAR_Machine.stOutletModule.iq_stStatus.q_xThirdPartySetupActive	AND
			NOT	VAR_Machine.stOutletModule.iq_stStatus.q_xThirdPartySetupDone	THEN
			uiThirdPartySetupStep	:=	400;
		END_IF

	400:
		xThirdPartySetupDone := TRUE;
END_CASE
END_STEP
ENTRY_ACTION
uiThirdPartySetupStep	:=	0;
xThirdPartySetupDone	:=	FALSE;
END_ACTION
EXIT_ACTION
VAR_Machine.stFillerModule.iq_stCmd.i_xThirdPartySetup 			:=	FALSE;
VAR_Machine.stFillerModule.iq_stParameters.i_uiAxisSelected		:=	CST_FirstFillerModuleAxis;

VAR_Machine.stOutletModule.iq_stCmd.i_xThirdPartySetup			:=	FALSE;
VAR_Machine.stOutletModule.iq_stParameters.i_uiAxisSelected		:=	CST_FirstOutletModuleAxis;

VAR_Machine.stInletModule.iq_stCmd.i_xThirdPartySetup			:=	FALSE;
VAR_Machine.stInletModule.iq_stParameters.i_uiAxisSelected		:=	CST_FirstInletModuleAxis;
END_ACTION
TRANSITION FROM ThirdPartySetup TO ThirdPartySetupExit:=
NOT xThirdPartySetupMode
END_TRANSITION
STEP ThirdPartySetupExit:
xExitStep				:= TRUE;
xThirdPartySetupDone	:= FALSE;
xThirdPartySetupActive	:= FALSE;
END_STEP
TRANSITION FROM ThirdPartySetupExit TO ModeSelection:=
xExitStep
END_TRANSITION
(* @SFCISJUMP := 'ModeSelection' *)
TRANSITION FROM ModeSelection TO InductionSetup:=
xInductionSetupMode
END_TRANSITION
STEP InductionSetup:
IF xInductionSetupDone OR xReactionActive THEN
	xInductionSetupMode	:= FALSE;
END_IF
```
